LIN {X 0,Y 656.687,Z 491.433,A -85,B 0,C 180,E1 28585.458,E2 28585.458} C_VEL
LIN {X 0,Y 656.704,Z 491.397,A -85,B 0,C 180,E1 28582.346,E2 28582.346} C_VEL
LIN {X 0,Y 656.703,Z 491.421,A -85,B 0,C 180,E1 28580.485,E2 28580.485} C_VEL
LIN {X 0,Y 655.757,Z 491.547,A -85,B 0,C 180,E1 28579.813,E2 28579.813} C_VEL
LIN {X 0,Y 649.317,Z 492.327,A -85,B 0,C 180,E1 28577.929,E2 28577.929} C_VEL
LIN {X 0,Y 648.761,Z 492.387,A -85,B 0,C 180,E1 28577.439,E2 28577.439} C_VEL
LIN {X 0,Y 648.764,Z 492.41,A -85,B 0,C 180,E1 28574.279,E2 28574.279} C_VEL
LIN {X 0,Y 648.798,Z 492.658,A -85,B 0,C 180,E1 28571.504,E2 28571.504} C_VEL
LIN {X 0,Y 657.705,Z 514.386,A -85,B 0,C 180,E1 28569.164,E2 28569.164} C_VEL
LIN {X 0,Y 662.553,Z 527.138,A -85,B 0,C 180,E1 28567.894,E2 28567.894} C_VEL
LIN {X 0,Y 660.274,Z 574.159,A -85,B 0,C 180,E1 28564.707,E2 28564.707} C_VEL
LIN {X 0,Y 658.321,Z 619.289,A -85,B 0,C 180,E1 28561.727,E2 28561.727} C_VEL
LIN {X 0,Y 657.32,Z 647.28,A -85,B 0,C 180,E1 28559.941,E2 28559.941} C_VEL
LIN {X 0,Y 661.313,Z 670.225,A -85,B 0,C 180,E1 28559.432,E2 28559.432} C_VEL
LIN {X 0,Y 659.221,Z 900.56,A -85,B 0,C 180,E1 28556.758,E2 28556.758} C_VEL
LIN {X 0,Y 658.59,Z 956.878,A -85,B 0,C 180,E1 28556.077,E2 28556.077} C_VEL
LIN {X 0,Y 657.927,Z 978.152,A -85,B 0,C 180,E1 28555.662,E2 28555.662} C_VEL
LIN {X 0,Y 657.104,Z 999.966,A -85,B 0,C 180,E1 28555.073,E2 28555.073} C_VEL
LIN {X 0,Y 656.193,Z 1019.608,A -85,B 0,C 180,E1 28554.389,E2 28554.389} C_VEL
LIN {X 0,Y 655.097,Z 1039.619,A -85,B 0,C 180,E1 28553.523,E2 28553.523} C_VEL
LIN {X 0,Y 653.941,Z 1059.736,A -85,B 0,C 180,E1 28552.473,E2 28552.473} C_VEL
LIN {X 0,Y 652.846,Z 1078.181,A -85,B 0,C 180,E1 28551.33,E2 28551.33} C_VEL
LIN {X 0,Y 651.725,Z 1096.211,A -85,B 0,C 180,E1 28550.006,E2 28550.006} C_VEL
LIN {X 0,Y 650.802,Z 1113.681,A -85,B 0,C 180,E1 28548.543,E2 28548.543} C_VEL
LIN {X 0,Y 650.064,Z 1128.76,A -85,B 0,C 180,E1 28547.084,E2 28547.084} C_VEL
LIN {X 0,Y 649.402,Z 1143.252,A -85,B 0,C 180,E1 28545.448,E2 28545.448} C_VEL
LIN {X 0,Y 648.879,Z 1155.499,A -85,B 0,C 180,E1 28543.818,E2 28543.818} C_VEL
LIN {X 0,Y 648.48,Z 1167.039,A -85,B 0,C 180,E1 28542.014,E2 28542.014} C_VEL
LIN {X 0,Y 648.221,Z 1176.646,A -85,B 0,C 180,E1 28540.217,E2 28540.217} C_VEL
LIN {X 0,Y 648.06,Z 1184.7,A -85,B 0,C 180,E1 28538.339,E2 28538.339} C_VEL
LIN {X 0,Y 647.959,Z 1191.273,A -85,B 0,C 180,E1 28536.379,E2 28536.379} C_VEL
LIN {X 0,Y 647.926,Z 1195.934,A -85,B 0,C 180,E1 28534.495,E2 28534.495} C_VEL
LIN {X 0,Y 647.913,Z 1198.843,A -85,B 0,C 180,E1 28532.654,E2 28532.654} C_VEL
LIN {X 0,Y 647.907,Z 1200.334,A -85,B 0,C 180,E1 28530.619,E2 28530.619} C_VEL
LIN {X 0,Y 647.902,Z 1200.184,A -85,B 0,C 180,E1 28528.762,E2 28528.762} C_VEL
LIN {X 0,Y 647.911,Z 1198.323,A -85,B 0,C 180,E1 28526.851,E2 28526.851} C_VEL
LIN {X 0,Y 647.927,Z 1194.711,A -85,B 0,C 180,E1 28524.865,E2 28524.865} C_VEL
LIN {X 0,Y 647.972,Z 1189.734,A -85,B 0,C 180,E1 28522.998,E2 28522.998} C_VEL
LIN {X 0,Y 648.084,Z 1182.936,A -85,B 0,C 180,E1 28521.125,E2 28521.125} C_VEL
LIN {X 0,Y 648.283,Z 1174.365,A -85,B 0,C 180,E1 28519.244,E2 28519.244} C_VEL
LIN {X 0,Y 648.58,Z 1164.395,A -85,B 0,C 180,E1 28517.446,E2 28517.446} C_VEL
LIN {X 0,Y 648.996,Z 1152.865,A -85,B 0,C 180,E1 28515.717,E2 28515.717} C_VEL
LIN {X 0,Y 649.521,Z 1140.155,A -85,B 0,C 180,E1 28514.097,E2 28514.097} C_VEL
LIN {X 0,Y 650.186,Z 1126.103,A -85,B 0,C 180,E1 28512.55,E2 28512.55} C_VEL
LIN {X 0,Y 650.967,Z 1110.603,A -85,B 0,C 180,E1 28511.09,E2 28511.09} C_VEL
LIN {X 0,Y 652.128,Z 1089.891,A -85,B 0,C 180,E1 28509.414,E2 28509.414} C_VEL
LIN {X 0,Y 653.168,Z 1072.447,A -85,B 0,C 180,E1 28508.21,E2 28508.21} C_VEL
LIN {X 0,Y 654.338,Z 1053.073,A -85,B 0,C 180,E1 28507.067,E2 28507.067} C_VEL
LIN {X 0,Y 655.454,Z 1033.69,A -85,B 0,C 180,E1 28506.109,E2 28506.109} C_VEL
LIN {X 0,Y 656.48,Z 1013.299,A -85,B 0,C 180,E1 28505.287,E2 28505.287} C_VEL
LIN {X 0,Y 657.466,Z 991.151,A -85,B 0,C 180,E1 28504.578,E2 28504.578} C_VEL
LIN {X 0,Y 658.227,Z 970.127,A -85,B 0,C 180,E1 28504.069,E2 28504.069} C_VEL
LIN {X 0,Y 658.733,Z 948.225,A -85,B 0,C 180,E1 28503.712,E2 28503.712} C_VEL
LIN {X 0,Y 660.553,Z 758.083,A -85,B 0,C 180,E1 28501.489,E2 28501.489} C_VEL
LIN {X 0,Y 661.13,Z 667.999,A -85,B 0,C 180,E1 28500.44,E2 28500.44} C_VEL
LIN {X 0,Y 657.249,Z 646.305,A -85,B 0,C 180,E1 28499.93,E2 28499.93} C_VEL
LIN {X 0,Y 659.188,Z 599.058,A -85,B 0,C 180,E1 28496.857,E2 28496.857} C_VEL
LIN {X 0,Y 661.229,Z 553.533,A -85,B 0,C 180,E1 28493.814,E2 28493.814} C_VEL
LIN {X 0,Y 662.53,Z 526.699,A -85,B 0,C 180,E1 28491.981,E2 28491.981} C_VEL
LIN {X 0,Y 654.583,Z 506.578,A -85,B 0,C 180,E1 28489.933,E2 28489.933} C_VEL
LIN {X 0,Y 648.804,Z 492.683,A -85,B 0,C 180,E1 28488.4,E2 28488.4} C_VEL
LIN {X 0,Y 648.764,Z 492.389,A -85,B 0,C 180,E1 28486.417,E2 28486.417} C_VEL
LIN {X 0,Y 648.737,Z 492.391,A -85,B 0,C 180,E1 28483.305,E2 28483.305} C_VEL
LIN {X 0,Y 648.771,Z 492.42,A -85,B 0,C 180,E1 28480.282,E2 28480.282} C_VEL
LIN {X 0,Y 648.738,Z 492.392,A -85,B 0,C 180,E1 28477.17,E2 28477.17} C_VEL
LIN {X 0,Y 648.767,Z 492.414,A -85,B 0,C 180,E1 28474.125,E2 28474.125} C_VEL
LIN {X 0,Y 648.738,Z 492.415,A -85,B 0,C 180,E1 28470.984,E2 28470.984} C_VEL
LIN {X 0,Y 648.77,Z 492.416,A -85,B 0,C 180,E1 28467.939,E2 28467.939} C_VEL
LIN {X 0,Y 648.735,Z 492.417,A -85,B 0,C 180,E1 28464.786,E2 28464.786} C_VEL
LIN {X 0,Y 648.773,Z 492.416,A -85,B 0,C 180,E1 28461.709,E2 28461.709} C_VEL
LIN {X 0,Y 648.733,Z 492.407,A -85,B 0,C 180,E1 28458.583,E2 28458.583} C_VEL
LIN {X 0,Y 648.767,Z 492.41,A -85,B 0,C 180,E1 28455.556,E2 28455.556} C_VEL
LIN {X 0,Y 648.735,Z 492.416,A -85,B 0,C 180,E1 28452.461,E2 28452.461} C_VEL
LIN {X 0,Y 648.765,Z 492.411,A -85,B 0,C 180,E1 28449.403,E2 28449.403} C_VEL
LIN {X 0,Y 648.732,Z 492.408,A -85,B 0,C 180,E1 28446.283,E2 28446.283} C_VEL
LIN {X 0,Y 648.76,Z 492.423,A -85,B 0,C 180,E1 28443.269,E2 28443.269} C_VEL
LIN {X 0,Y 648.729,Z 492.412,A -85,B 0,C 180,E1 28440.088,E2 28440.088} C_VEL
LIN {X 0,Y 648.76,Z 492.41,A -85,B 0,C 180,E1 28437.085,E2 28437.085} C_VEL
LIN {X 0,Y 648.729,Z 492.416,A -85,B 0,C 180,E1 28433.895,E2 28433.895} C_VEL
LIN {X 0,Y 648.755,Z 492.41,A -85,B 0,C 180,E1 28430.955,E2 28430.955} C_VEL
LIN {X 0,Y 648.732,Z 492.407,A -85,B 0,C 180,E1 28427.81,E2 28427.81} C_VEL
LIN {X 0,Y 648.741,Z 492.422,A -85,B 0,C 180,E1 28424.902,E2 28424.902} C_VEL
LIN {X 0,Y 648.735,Z 492.415,A -85,B 0,C 180,E1 28421.674,E2 28421.674} C_VEL
LIN {X 0,Y 648.736,Z 492.411,A -85,B 0,C 180,E1 28418.764,E2 28418.764} C_VEL
LIN {X 0,Y 648.733,Z 492.407,A -85,B 0,C 180,E1 28415.505,E2 28415.505} C_VEL
LIN {X 0,Y 648.735,Z 492.423,A -85,B 0,C 180,E1 28412.592,E2 28412.592} C_VEL
LIN {X 0,Y 648.733,Z 492.416,A -85,B 0,C 180,E1 28409.318,E2 28409.318} C_VEL
LIN {X 0,Y 648.73,Z 492.385,A -85,B 0,C 180,E1 28406.404,E2 28406.404} C_VEL
LIN {X 0,Y 648.733,Z 492.417,A -85,B 0,C 180,E1 28403.161,E2 28403.161} C_VEL
LIN {X 0,Y 648.724,Z 492.39,A -85,B 0,C 180,E1 28400.272,E2 28400.272} C_VEL
LIN {X 0,Y 648.737,Z 492.398,A -85,B 0,C 180,E1 28397.058,E2 28397.058} C_VEL
LIN {X 0,Y 648.722,Z 492.426,A -85,B 0,C 180,E1 28394.159,E2 28394.159} C_VEL
LIN {X 0,Y 648.764,Z 492.635,A -85,B 0,C 180,E1 28391.933,E2 28391.933} C_VEL
LIN {X 0,Y 653.027,Z 502.897,A -85,B 0,C 180,E1 28390.827,E2 28390.827} C_VEL
LIN {X 0,Y 660.861,Z 521.597,A -85,B 0,C 180,E1 28388.95,E2 28388.95} C_VEL
LIN {X 0,Y 663.163,Z 527.795,A -85,B 0,C 180,E1 28388.368,E2 28388.368} C_VEL
LIN {X 0,Y 663.076,Z 532.792,A -85,B 0,C 180,E1 28388.071,E2 28388.071} C_VEL
LIN {X 0,Y 666.748,Z 551.518,A -85,B 0,C 180,E1 28387.604,E2 28387.604} C_VEL
LIN {X 0,Y 664.218,Z 791.043,A -85,B 0,C 180,E1 28384.694,E2 28384.694} C_VEL
LIN {X 0,Y 663.116,Z 920.342,A -85,B 0,C 180,E1 28383.165,E2 28383.165} C_VEL
LIN {X 0,Y 662.457,Z 946.043,A -85,B 0,C 180,E1 28382.706,E2 28382.706} C_VEL
LIN {X 0,Y 661.756,Z 967.211,A -85,B 0,C 180,E1 28382.199,E2 28382.199} C_VEL
LIN {X 0,Y 660.811,Z 989.286,A -85,B 0,C 180,E1 28381.518,E2 28381.518} C_VEL
LIN {X 0,Y 659.621,Z 1011.361,A -85,B 0,C 180,E1 28380.668,E2 28380.668} C_VEL
LIN {X 0,Y 658.378,Z 1033.294,A -85,B 0,C 180,E1 28379.675,E2 28379.675} C_VEL
LIN {X 0,Y 656.934,Z 1055.135,A -85,B 0,C 180,E1 28378.499,E2 28378.499} C_VEL
LIN {X 0,Y 655.615,Z 1075.664,A -85,B 0,C 180,E1 28377.227,E2 28377.227} C_VEL
LIN {X 0,Y 654.266,Z 1095.229,A -85,B 0,C 180,E1 28375.82,E2 28375.82} C_VEL
LIN {X 0,Y 653.063,Z 1113.21,A -85,B 0,C 180,E1 28374.357,E2 28374.357} C_VEL
LIN {X 0,Y 651.925,Z 1130.611,A -85,B 0,C 180,E1 28372.736,E2 28372.736} C_VEL
LIN {X 0,Y 650.985,Z 1145.636,A -85,B 0,C 180,E1 28371.158,E2 28371.158} C_VEL
LIN {X 0,Y 650.057,Z 1162.032,A -85,B 0,C 180,E1 28369.19,E2 28369.19} C_VEL
LIN {X 0,Y 649.427,Z 1174.524,A -85,B 0,C 180,E1 28367.471,E2 28367.471} C_VEL
LIN {X 0,Y 648.841,Z 1187.771,A -85,B 0,C 180,E1 28365.37,E2 28365.37} C_VEL
LIN {X 0,Y 648.474,Z 1197.565,A -85,B 0,C 180,E1 28363.554,E2 28363.554} C_VEL
LIN {X 0,Y 648.202,Z 1207.125,A -85,B 0,C 180,E1 28361.478,E2 28361.478} C_VEL
LIN {X 0,Y 648.054,Z 1214.515,A -85,B 0,C 180,E1 28359.502,E2 28359.502} C_VEL
LIN {X 0,Y 647.94,Z 1220.508,A -85,B 0,C 180,E1 28357.537,E2 28357.537} C_VEL
LIN {X 0,Y 647.901,Z 1225.336,A -85,B 0,C 180,E1 28355.402,E2 28355.402} C_VEL
LIN {X 0,Y 647.912,Z 1228.238,A -85,B 0,C 180,E1 28353.539,E2 28353.539} C_VEL
LIN {X 0,Y 647.904,Z 1230.169,A -85,B 0,C 180,E1 28351.326,E2 28351.326} C_VEL
LIN {X 0,Y 647.883,Z 1230.351,A -85,B 0,C 180,E1 28349.381,E2 28349.381} C_VEL
LIN {X 0,Y 647.899,Z 1229.361,A -85,B 0,C 180,E1 28347.523,E2 28347.523} C_VEL
LIN {X 0,Y 647.915,Z 1226.609,A -85,B 0,C 180,E1 28345.309,E2 28345.309} C_VEL
LIN {X 0,Y 647.941,Z 1222.896,A -85,B 0,C 180,E1 28343.443,E2 28343.443} C_VEL
LIN {X 0,Y 648.004,Z 1217.711,A -85,B 0,C 180,E1 28341.482,E2 28341.482} C_VEL
LIN {X 0,Y 648.138,Z 1210.307,A -85,B 0,C 180,E1 28339.331,E2 28339.331} C_VEL
LIN {X 0,Y 648.327,Z 1202.569,A -85,B 0,C 180,E1 28337.49,E2 28337.49} C_VEL
LIN {X 0,Y 648.682,Z 1191.897,A -85,B 0,C 180,E1 28335.358,E2 28335.358} C_VEL
LIN {X 0,Y 649.116,Z 1181.124,A -85,B 0,C 180,E1 28333.535,E2 28333.535} C_VEL
LIN {X 0,Y 649.762,Z 1168.129,A -85,B 0,C 180,E1 28331.612,E2 28331.612} C_VEL
LIN {X 0,Y 650.527,Z 1153.627,A -85,B 0,C 180,E1 28329.768,E2 28329.768} C_VEL
LIN {X 0,Y 651.499,Z 1137.653,A -85,B 0,C 180,E1 28327.971,E2 28327.971} C_VEL
LIN {X 0,Y 652.547,Z 1120.834,A -85,B 0,C 180,E1 28326.331,E2 28326.331} C_VEL
LIN {X 0,Y 653.8,Z 1102.507,A -85,B 0,C 180,E1 28324.743,E2 28324.743} C_VEL
LIN {X 0,Y 655.079,Z 1083.079,A -85,B 0,C 180,E1 28323.288,E2 28323.288} C_VEL
LIN {X 0,Y 656.509,Z 1062.412,A -85,B 0,C 180,E1 28321.927,E2 28321.927} C_VEL
LIN {X 0,Y 657.802,Z 1041.566,A -85,B 0,C 180,E1 28320.752,E2 28320.752} C_VEL
LIN {X 0,Y 659.216,Z 1019.235,A -85,B 0,C 180,E1 28319.664,E2 28319.664} C_VEL
LIN {X 0,Y 660.407,Z 996.993,A -85,B 0,C 180,E1 28318.765,E2 28318.765} C_VEL
LIN {X 0,Y 661.384,Z 976.854,A -85,B 0,C 180,E1 28318.08,E2 28318.08} C_VEL
LIN {X 0,Y 662.227,Z 952.701,A -85,B 0,C 180,E1 28317.437,E2 28317.437} C_VEL
LIN {X 0,Y 662.87,Z 930.275,A -85,B 0,C 180,E1 28316.993,E2 28316.993} C_VEL
LIN {X 0,Y 663.356,Z 902.806,A -85,B 0,C 180,E1 28316.61,E2 28316.61} C_VEL
LIN {X 0,Y 665.273,Z 677.94,A -85,B 0,C 180,E1 28313.952,E2 28313.952} C_VEL
LIN {X 0,Y 666.596,Z 549.747,A -85,B 0,C 180,E1 28312.364,E2 28312.364} C_VEL
LIN {X 0,Y 662.988,Z 531.826,A -85,B 0,C 180,E1 28311.889,E2 28311.889} C_VEL
LIN {X 0,Y 663.187,Z 527.295,A -85,B 0,C 180,E1 28311.6,E2 28311.6} C_VEL
LIN {X 0,Y 654.413,Z 506.148,A -85,B 0,C 180,E1 28309.508,E2 28309.508} C_VEL
LIN {X 0,Y 648.773,Z 492.677,A -85,B 0,C 180,E1 28308.078,E2 28308.078} C_VEL
LIN {X 0,Y 648.772,Z 492.403,A -85,B 0,C 180,E1 28306.579,E2 28306.579} C_VEL
LIN {X 0,Y 648.71,Z 492.393,A -85,B 0,C 180,E1 28303.55,E2 28303.55} C_VEL
LIN {X 0,Y 648.77,Z 492.407,A -85,B 0,C 180,E1 28300.571,E2 28300.571} C_VEL
LIN {X 0,Y 648.718,Z 492.415,A -85,B 0,C 180,E1 28297.462,E2 28297.462} C_VEL
LIN {X 0,Y 648.755,Z 492.399,A -85,B 0,C 180,E1 28294.554,E2 28294.554} C_VEL
LIN {X 0,Y 648.724,Z 492.417,A -85,B 0,C 180,E1 28291.366,E2 28291.366} C_VEL
LIN {X 0,Y 648.751,Z 492.409,A -85,B 0,C 180,E1 28288.441,E2 28288.441} C_VEL
LIN {X 0,Y 648.732,Z 492.411,A -85,B 0,C 180,E1 28285.274,E2 28285.274} C_VEL
LIN {X 0,Y 648.741,Z 492.415,A -85,B 0,C 180,E1 28282.372,E2 28282.372} C_VEL
LIN {X 0,Y 648.738,Z 492.421,A -85,B 0,C 180,E1 28279.131,E2 28279.131} C_VEL
LIN {X 0,Y 648.742,Z 492.408,A -85,B 0,C 180,E1 28276.199,E2 28276.199} C_VEL
LIN {X 0,Y 648.742,Z 492.41,A -85,B 0,C 180,E1 28273.004,E2 28273.004} C_VEL
LIN {X 0,Y 648.747,Z 492.414,A -85,B 0,C 180,E1 28269.992,E2 28269.992} C_VEL
LIN {X 0,Y 648.746,Z 492.42,A -85,B 0,C 180,E1 28266.816,E2 28266.816} C_VEL
LIN {X 0,Y 648.747,Z 492.405,A -85,B 0,C 180,E1 28263.8,E2 28263.8} C_VEL
LIN {X 0,Y 648.747,Z 492.417,A -85,B 0,C 180,E1 28260.618,E2 28260.618} C_VEL
LIN {X 0,Y 648.75,Z 492.41,A -85,B 0,C 180,E1 28257.615,E2 28257.615} C_VEL
LIN {X 0,Y 648.745,Z 492.409,A -85,B 0,C 180,E1 28254.428,E2 28254.428} C_VEL
LIN {X 0,Y 648.756,Z 492.413,A -85,B 0,C 180,E1 28251.402,E2 28251.402} C_VEL
LIN {X 0,Y 648.743,Z 492.422,A -85,B 0,C 180,E1 28248.171,E2 28248.171} C_VEL
LIN {X 0,Y 648.77,Z 492.401,A -85,B 0,C 180,E1 28245.084,E2 28245.084} C_VEL
LIN {X 0,Y 648.743,Z 492.412,A -85,B 0,C 180,E1 28241.953,E2 28241.953} C_VEL
LIN {X 0,Y 648.77,Z 492.413,A -85,B 0,C 180,E1 28238.86,E2 28238.86} C_VEL
LIN {X 0,Y 648.741,Z 492.421,A -85,B 0,C 180,E1 28235.699,E2 28235.699} C_VEL
LIN {X 0,Y 648.766,Z 492.406,A -85,B 0,C 180,E1 28232.659,E2 28232.659} C_VEL
LIN {X 0,Y 648.743,Z 492.415,A -85,B 0,C 180,E1 28229.53,E2 28229.53} C_VEL
LIN {X 0,Y 648.766,Z 492.408,A -85,B 0,C 180,E1 28226.488,E2 28226.488} C_VEL
LIN {X 0,Y 648.744,Z 492.399,A -85,B 0,C 180,E1 28223.382,E2 28223.382} C_VEL
LIN {X 0,Y 648.768,Z 492.41,A -85,B 0,C 180,E1 28220.268,E2 28220.268} C_VEL
LIN {X 0,Y 648.761,Z 492.387,A -85,B 0,C 180,E1 28217.439,E2 28217.439} C_VEL
LIN {X 0,Y 647.741,Z 492.518,A -85,B 0,C 180,E1 28216.759,E2 28216.759} C_VEL
LIN {X 0,Y 641.323,Z 493.349,A -85,B 0,C 180,E1 28214.852,E2 28214.852} C_VEL
LIN {X 0,Y 640.821,Z 493.4,A -85,B 0,C 180,E1 28214.356,E2 28214.356} C_VEL
LIN {X 0,Y 640.86,Z 493.629,A -85,B 0,C 180,E1 28212.067,E2 28212.067} C_VEL
LIN {X 0,Y 645.223,Z 504.16,A -85,B 0,C 180,E1 28210.865,E2 28210.865} C_VEL
LIN {X 0,Y 653.936,Z 525.683,A -85,B 0,C 180,E1 28208.596,E2 28208.596} C_VEL
LIN {X 0,Y 655.646,Z 530.796,A -85,B 0,C 180,E1 28208.101,E2 28208.101} C_VEL
LIN {X 0,Y 653.146,Z 578.763,A -85,B 0,C 180,E1 28204.82,E2 28204.82} C_VEL
LIN {X 0,Y 651.038,Z 624.276,A -85,B 0,C 180,E1 28201.788,E2 28201.788} C_VEL
LIN {X 0,Y 650.196,Z 646.313,A -85,B 0,C 180,E1 28200.37,E2 28200.37} C_VEL
LIN {X 0,Y 654.607,Z 671.415,A -85,B 0,C 180,E1 28199.802,E2 28199.802} C_VEL
LIN {X 0,Y 652.343,Z 919.767,A -85,B 0,C 180,E1 28196.919,E2 28196.919} C_VEL
LIN {X 0,Y 651.813,Z 958.309,A -85,B 0,C 180,E1 28196.435,E2 28196.435} C_VEL
LIN {X 0,Y 651.111,Z 979.366,A -85,B 0,C 180,E1 28196.015,E2 28196.015} C_VEL
LIN {X 0,Y 650.23,Z 1000.616,A -85,B 0,C 180,E1 28195.43,E2 28195.43} C_VEL
LIN {X 0,Y 649.223,Z 1020.828,A -85,B 0,C 180,E1 28194.717,E2 28194.717} C_VEL
LIN {X 0,Y 648.016,Z 1040.55,A -85,B 0,C 180,E1 28193.844,E2 28193.844} C_VEL
LIN {X 0,Y 646.736,Z 1060.42,A -85,B 0,C 180,E1 28192.785,E2 28192.785} C_VEL
LIN {X 0,Y 645.476,Z 1079.395,A -85,B 0,C 180,E1 28191.586,E2 28191.586} C_VEL
LIN {X 0,Y 644.291,Z 1096.703,A -85,B 0,C 180,E1 28190.294,E2 28190.294} C_VEL
LIN {X 0,Y 643.211,Z 1113.172,A -85,B 0,C 180,E1 28188.864,E2 28188.864} C_VEL
LIN {X 0,Y 642.272,Z 1128.765,A -85,B 0,C 180,E1 28187.298,E2 28187.298} C_VEL
LIN {X 0,Y 641.549,Z 1143.255,A -85,B 0,C 180,E1 28185.642,E2 28185.642} C_VEL
LIN {X 0,Y 640.981,Z 1155.501,A -85,B 0,C 180,E1 28183.992,E2 28183.992} C_VEL
LIN {X 0,Y 640.54,Z 1167.041,A -85,B 0,C 180,E1 28182.165,E2 28182.165} C_VEL
LIN {X 0,Y 640.254,Z 1176.649,A -85,B 0,C 180,E1 28180.346,E2 28180.346} C_VEL
LIN {X 0,Y 640.078,Z 1184.703,A -85,B 0,C 180,E1 28178.444,E2 28178.444} C_VEL
LIN {X 0,Y 639.962,Z 1191.274,A -85,B 0,C 180,E1 28176.459,E2 28176.459} C_VEL
LIN {X 0,Y 639.925,Z 1195.988,A -85,B 0,C 180,E1 28174.521,E2 28174.521} C_VEL
LIN {X 0,Y 639.912,Z 1198.843,A -85,B 0,C 180,E1 28172.687,E2 28172.687} C_VEL
LIN {X 0,Y 639.907,Z 1200.334,A -85,B 0,C 180,E1 28170.627,E2 28170.627} C_VEL
LIN {X 0,Y 639.902,Z 1200.184,A -85,B 0,C 180,E1 28168.747,E2 28168.747} C_VEL
LIN {X 0,Y 639.911,Z 1198.349,A -85,B 0,C 180,E1 28166.833,E2 28166.833} C_VEL
LIN {X 0,Y 639.931,Z 1194.71,A -85,B 0,C 180,E1 28164.801,E2 28164.801} C_VEL
LIN {X 0,Y 639.982,Z 1189.732,A -85,B 0,C 180,E1 28162.91,E2 28162.91} C_VEL
LIN {X 0,Y 640.103,Z 1182.934,A -85,B 0,C 180,E1 28161.013,E2 28161.013} C_VEL
LIN {X 0,Y 640.319,Z 1174.362,A -85,B 0,C 180,E1 28159.109,E2 28159.109} C_VEL
LIN {X 0,Y 640.651,Z 1164.361,A -85,B 0,C 180,E1 28157.283,E2 28157.283} C_VEL
LIN {X 0,Y 641.1,Z 1152.947,A -85,B 0,C 180,E1 28155.55,E2 28155.55} C_VEL
LIN {X 0,Y 641.681,Z 1140.149,A -85,B 0,C 180,E1 28153.898,E2 28153.898} C_VEL
LIN {X 0,Y 642.459,Z 1125.255,A -85,B 0,C 180,E1 28152.24,E2 28152.24} C_VEL
LIN {X 0,Y 643.442,Z 1109.685,A -85,B 0,C 180,E1 28150.719,E2 28150.719} C_VEL
LIN {X 0,Y 644.535,Z 1093.11,A -85,B 0,C 180,E1 28149.334,E2 28149.334} C_VEL
LIN {X 0,Y 645.789,Z 1074.445,A -85,B 0,C 180,E1 28147.995,E2 28147.995} C_VEL
LIN {X 0,Y 647.09,Z 1055.489,A -85,B 0,C 180,E1 28146.839,E2 28146.839} C_VEL
LIN {X 0,Y 648.263,Z 1036.558,A -85,B 0,C 180,E1 28145.875,E2 28145.875} C_VEL
LIN {X 0,Y 649.469,Z 1015.731,A -85,B 0,C 180,E1 28145.002,E2 28145.002} C_VEL
LIN {X 0,Y 650.499,Z 995.068,A -85,B 0,C 180,E1 28144.307,E2 28144.307} C_VEL
LIN {X 0,Y 651.297,Z 974.495,A -85,B 0,C 180,E1 28143.785,E2 28143.785} C_VEL
LIN {X 0,Y 651.929,Z 951.776,A -85,B 0,C 180,E1 28143.38,E2 28143.38} C_VEL
LIN {X 0,Y 653.583,Z 787.252,A -85,B 0,C 180,E1 28141.444,E2 28141.444} C_VEL
LIN {X 0,Y 654.426,Z 669.373,A -85,B 0,C 180,E1 28140.073,E2 28140.073} C_VEL
LIN {X 0,Y 650.137,Z 645.401,A -85,B 0,C 180,E1 28139.502,E2 28139.502} C_VEL
LIN {X 0,Y 652.213,Z 598.269,A -85,B 0,C 180,E1 28136.398,E2 28136.398} C_VEL
LIN {X 0,Y 654.413,Z 553.495,A -85,B 0,C 180,E1 28133.371,E2 28133.371} C_VEL
LIN {X 0,Y 655.594,Z 529.964,A -85,B 0,C 180,E1 28131.743,E2 28131.743} C_VEL
LIN {X 0,Y 646.809,Z 507.86,A -85,B 0,C 180,E1 28129.447,E2 28129.447} C_VEL
LIN {X 0,Y 640.888,Z 493.793,A -85,B 0,C 180,E1 28127.868,E2 28127.868} C_VEL
LIN {X 0,Y 640.794,Z 493.374,A -85,B 0,C 180,E1 28127.303,E2 28127.303} C_VEL
LIN {X 0,Y 640.826,Z 493.394,A -85,B 0,C 180,E1 28124.224,E2 28124.224} C_VEL
LIN {X 0,Y 640.795,Z 493.403,A -85,B 0,C 180,E1 28121.093,E2 28121.093} C_VEL
LIN {X 0,Y 640.824,Z 493.37,A -85,B 0,C 180,E1 28118.049,E2 28118.049} C_VEL
LIN {X 0,Y 640.794,Z 493.408,A -85,B 0,C 180,E1 28114.936,E2 28114.936} C_VEL
LIN {X 0,Y 640.828,Z 493.409,A -85,B 0,C 180,E1 28111.921,E2 28111.921} C_VEL
LIN {X 0,Y 640.795,Z 493.406,A -85,B 0,C 180,E1 28108.827,E2 28108.827} C_VEL
LIN {X 0,Y 640.83,Z 493.403,A -85,B 0,C 180,E1 28105.806,E2 28105.806} C_VEL
LIN {X 0,Y 640.793,Z 493.395,A -85,B 0,C 180,E1 28102.67,E2 28102.67} C_VEL
LIN {X 0,Y 640.829,Z 493.398,A -85,B 0,C 180,E1 28099.696,E2 28099.696} C_VEL
LIN {X 0,Y 640.798,Z 493.405,A -85,B 0,C 180,E1 28096.592,E2 28096.592} C_VEL
LIN {X 0,Y 640.828,Z 493.402,A -85,B 0,C 180,E1 28093.536,E2 28093.536} C_VEL
LIN {X 0,Y 640.796,Z 493.392,A -85,B 0,C 180,E1 28090.428,E2 28090.428} C_VEL
LIN {X 0,Y 640.822,Z 493.408,A -85,B 0,C 180,E1 28087.441,E2 28087.441} C_VEL
LIN {X 0,Y 640.799,Z 493.403,A -85,B 0,C 180,E1 28084.295,E2 28084.295} C_VEL
LIN {X 0,Y 640.818,Z 493.397,A -85,B 0,C 180,E1 28081.252,E2 28081.252} C_VEL
LIN {X 0,Y 640.797,Z 493.403,A -85,B 0,C 180,E1 28078.122,E2 28078.122} C_VEL
LIN {X 0,Y 640.816,Z 493.403,A -85,B 0,C 180,E1 28075.077,E2 28075.077} C_VEL
LIN {X 0,Y 640.794,Z 493.391,A -85,B 0,C 180,E1 28071.927,E2 28071.927} C_VEL
LIN {X 0,Y 640.813,Z 493.41,A -85,B 0,C 180,E1 28068.935,E2 28068.935} C_VEL
LIN {X 0,Y 640.79,Z 493.405,A -85,B 0,C 180,E1 28065.727,E2 28065.727} C_VEL
LIN {X 0,Y 640.809,Z 493.398,A -85,B 0,C 180,E1 28062.754,E2 28062.754} C_VEL
LIN {X 0,Y 640.79,Z 493.398,A -85,B 0,C 180,E1 28059.541,E2 28059.541} C_VEL
LIN {X 0,Y 640.803,Z 493.411,A -85,B 0,C 180,E1 28056.651,E2 28056.651} C_VEL
LIN {X 0,Y 640.793,Z 493.406,A -85,B 0,C 180,E1 28053.39,E2 28053.39} C_VEL
LIN {X 0,Y 640.801,Z 493.406,A -85,B 0,C 180,E1 28050.457,E2 28050.457} C_VEL
LIN {X 0,Y 640.787,Z 493.375,A -85,B 0,C 180,E1 28047.217,E2 28047.217} C_VEL
LIN {X 0,Y 640.799,Z 493.406,A -85,B 0,C 180,E1 28044.297,E2 28044.297} C_VEL
LIN {X 0,Y 640.783,Z 493.371,A -85,B 0,C 180,E1 28041.035,E2 28041.035} C_VEL
LIN {X 0,Y 640.789,Z 493.414,A -85,B 0,C 180,E1 28038.218,E2 28038.218} C_VEL
LIN {X 0,Y 640.795,Z 493.392,A -85,B 0,C 180,E1 28034.978,E2 28034.978} C_VEL
LIN {X 0,Y 640.799,Z 493.589,A -85,B 0,C 180,E1 28032.502,E2 28032.502} C_VEL
LIN {X 0,Y 641.926,Z 496.622,A -85,B 0,C 180,E1 28032.146,E2 28032.146} C_VEL
LIN {X 0,Y 650.144,Z 515.394,A -85,B 0,C 180,E1 28030.149,E2 28030.149} C_VEL
LIN {X 0,Y 656.315,Z 530.866,A -85,B 0,C 180,E1 28028.623,E2 28028.623} C_VEL
LIN {X 0,Y 656.391,Z 534.026,A -85,B 0,C 180,E1 28028.455,E2 28028.455} C_VEL
LIN {X 0,Y 660.104,Z 553.023,A -85,B 0,C 180,E1 28027.975,E2 28027.975} C_VEL
LIN {X 0,Y 657.263,Z 788.968,A -85,B 0,C 180,E1 28025.06,E2 28025.06} C_VEL
LIN {X 0,Y 655.972,Z 920.648,A -85,B 0,C 180,E1 28023.477,E2 28023.477} C_VEL
LIN {X 0,Y 655.269,Z 946.268,A -85,B 0,C 180,E1 28023.013,E2 28023.013} C_VEL
LIN {X 0,Y 654.509,Z 967.887,A -85,B 0,C 180,E1 28022.488,E2 28022.488} C_VEL
LIN {X 0,Y 653.447,Z 993.177,A -85,B 0,C 180,E1 28021.703,E2 28021.703} C_VEL
LIN {X 0,Y 652.476,Z 1013.342,A -85,B 0,C 180,E1 28020.939,E2 28020.939} C_VEL
LIN {X 0,Y 651.301,Z 1033.298,A -85,B 0,C 180,E1 28020.031,E2 28020.031} C_VEL
LIN {X 0,Y 649.752,Z 1055.13,A -85,B 0,C 180,E1 28018.844,E2 28018.844} C_VEL
LIN {X 0,Y 648.312,Z 1075.667,A -85,B 0,C 180,E1 28017.56,E2 28017.56} C_VEL
LIN {X 0,Y 646.863,Z 1095.227,A -85,B 0,C 180,E1 28016.137,E2 28016.137} C_VEL
LIN {X 0,Y 645.554,Z 1113.071,A -85,B 0,C 180,E1 28014.671,E2 28014.671} C_VEL
LIN {X 0,Y 644.312,Z 1130.61,A -85,B 0,C 180,E1 28013.02,E2 28013.02} C_VEL
LIN {X 0,Y 643.278,Z 1145.866,A -85,B 0,C 180,E1 28011.398,E2 28011.398} C_VEL
LIN {X 0,Y 642.296,Z 1161.824,A -85,B 0,C 180,E1 28009.459,E2 28009.459} C_VEL
LIN {X 0,Y 641.577,Z 1174.522,A -85,B 0,C 180,E1 28007.692,E2 28007.692} C_VEL
LIN {X 0,Y 640.935,Z 1187.772,A -85,B 0,C 180,E1 28005.564,E2 28005.564} C_VEL
LIN {X 0,Y 640.537,Z 1197.564,A -85,B 0,C 180,E1 28003.725,E2 28003.725} C_VEL
LIN {X 0,Y 640.242,Z 1207.126,A -85,B 0,C 180,E1 28001.622,E2 28001.622} C_VEL
LIN {X 0,Y 640.062,Z 1214.515,A -85,B 0,C 180,E1 27999.622,E2 27999.622} C_VEL
LIN {X 0,Y 639.95,Z 1220.508,A -85,B 0,C 180,E1 27997.632,E2 27997.632} C_VEL
LIN {X 0,Y 639.905,Z 1225.336,A -85,B 0,C 180,E1 27995.469,E2 27995.469} C_VEL
LIN {X 0,Y 639.912,Z 1228.238,A -85,B 0,C 180,E1 27993.583,E2 27993.583} C_VEL
LIN {X 0,Y 639.903,Z 1230.169,A -85,B 0,C 180,E1 27991.343,E2 27991.343} C_VEL
LIN {X 0,Y 639.883,Z 1230.35,A -85,B 0,C 180,E1 27989.373,E2 27989.373} C_VEL
LIN {X 0,Y 639.897,Z 1229.361,A -85,B 0,C 180,E1 27987.492,E2 27987.492} C_VEL
LIN {X 0,Y 639.912,Z 1226.61,A -85,B 0,C 180,E1 27985.25,E2 27985.25} C_VEL
LIN {X 0,Y 639.945,Z 1222.896,A -85,B 0,C 180,E1 27983.361,E2 27983.361} C_VEL
LIN {X 0,Y 640.009,Z 1217.711,A -85,B 0,C 180,E1 27981.374,E2 27981.374} C_VEL
LIN {X 0,Y 640.157,Z 1210.31,A -85,B 0,C 180,E1 27979.197,E2 27979.197} C_VEL
LIN {X 0,Y 640.369,Z 1202.753,A -85,B 0,C 180,E1 27977.374,E2 27977.374} C_VEL
LIN {X 0,Y 640.747,Z 1192.41,A -85,B 0,C 180,E1 27975.265,E2 27975.265} C_VEL
LIN {X 0,Y 641.239,Z 1181.123,A -85,B 0,C 180,E1 27973.327,E2 27973.327} C_VEL
LIN {X 0,Y 641.945,Z 1168.128,A -85,B 0,C 180,E1 27971.38,E2 27971.38} C_VEL
LIN {X 0,Y 642.79,Z 1153.625,A -85,B 0,C 180,E1 27969.514,E2 27969.514} C_VEL
LIN {X 0,Y 643.823,Z 1138.007,A -85,B 0,C 180,E1 27967.733,E2 27967.733} C_VEL
LIN {X 0,Y 644.994,Z 1120.834,A -85,B 0,C 180,E1 27966.037,E2 27966.037} C_VEL
LIN {X 0,Y 646.34,Z 1102.508,A -85,B 0,C 180,E1 27964.431,E2 27964.431} C_VEL
LIN {X 0,Y 647.747,Z 1083.049,A -85,B 0,C 180,E1 27962.96,E2 27962.96} C_VEL
LIN {X 0,Y 649.224,Z 1063.177,A -85,B 0,C 180,E1 27961.633,E2 27961.633} C_VEL
LIN {X 0,Y 650.635,Z 1042.29,A -85,B 0,C 180,E1 27960.439,E2 27960.439} C_VEL
LIN {X 0,Y 651.976,Z 1022.236,A -85,B 0,C 180,E1 27959.444,E2 27959.444} C_VEL
LIN {X 0,Y 653.157,Z 999.802,A -85,B 0,C 180,E1 27958.533,E2 27958.533} C_VEL
LIN {X 0,Y 654.077,Z 978.978,A -85,B 0,C 180,E1 27957.835,E2 27957.835} C_VEL
LIN {X 0,Y 654.974,Z 955.303,A -85,B 0,C 180,E1 27957.185,E2 27957.185} C_VEL
LIN {X 0,Y 655.672,Z 931.683,A -85,B 0,C 180,E1 27956.703,E2 27956.703} C_VEL
LIN {X 0,Y 656.203,Z 906.757,A -85,B 0,C 180,E1 27956.336,E2 27956.336} C_VEL
LIN {X 0,Y 658.409,Z 681.268,A -85,B 0,C 180,E1 27953.629,E2 27953.629} C_VEL
LIN {X 0,Y 659.962,Z 551.351,A -85,B 0,C 180,E1 27951.994,E2 27951.994} C_VEL
LIN {X 0,Y 656.245,Z 532.953,A -85,B 0,C 180,E1 27951.506,E2 27951.506} C_VEL
LIN {X 0,Y 656.21,Z 530.422,A -85,B 0,C 180,E1 27951.339,E2 27951.339} C_VEL
LIN {X 0,Y 646.982,Z 508.07,A -85,B 0,C 180,E1 27949.09,E2 27949.09} C_VEL
LIN {X 0,Y 640.811,Z 493.667,A -85,B 0,C 180,E1 27947.517,E2 27947.517} C_VEL
LIN {X 0,Y 640.809,Z 493.407,A -85,B 0,C 180,E1 27946.128,E2 27946.128} C_VEL
LIN {X 0,Y 640.777,Z 493.382,A -85,B 0,C 180,E1 27943.223,E2 27943.223} C_VEL
LIN {X 0,Y 640.829,Z 493.38,A -85,B 0,C 180,E1 27940.122,E2 27940.122} C_VEL
LIN {X 0,Y 640.779,Z 493.408,A -85,B 0,C 180,E1 27937.122,E2 27937.122} C_VEL
LIN {X 0,Y 640.827,Z 493.372,A -85,B 0,C 180,E1 27934.055,E2 27934.055} C_VEL
LIN {X 0,Y 640.778,Z 493.407,A -85,B 0,C 180,E1 27931.058,E2 27931.058} C_VEL
LIN {X 0,Y 640.834,Z 493.396,A -85,B 0,C 180,E1 27928.113,E2 27928.113} C_VEL
LIN {X 0,Y 640.781,Z 493.399,A -85,B 0,C 180,E1 27925.016,E2 27925.016} C_VEL
LIN {X 0,Y 640.836,Z 493.404,A -85,B 0,C 180,E1 27921.992,E2 27921.992} C_VEL
LIN {X 0,Y 640.787,Z 493.409,A -85,B 0,C 180,E1 27918.939,E2 27918.939} C_VEL
LIN {X 0,Y 640.826,Z 493.396,A -85,B 0,C 180,E1 27915.939,E2 27915.939} C_VEL
LIN {X 0,Y 640.789,Z 493.397,A -85,B 0,C 180,E1 27912.782,E2 27912.782} C_VEL
LIN {X 0,Y 640.825,Z 493.402,A -85,B 0,C 180,E1 27909.792,E2 27909.792} C_VEL
LIN {X 0,Y 640.793,Z 493.409,A -85,B 0,C 180,E1 27906.631,E2 27906.631} C_VEL
LIN {X 0,Y 640.825,Z 493.392,A -85,B 0,C 180,E1 27903.578,E2 27903.578} C_VEL
LIN {X 0,Y 640.795,Z 493.404,A -85,B 0,C 180,E1 27900.447,E2 27900.447} C_VEL
LIN {X 0,Y 640.826,Z 493.398,A -85,B 0,C 180,E1 27897.407,E2 27897.407} C_VEL
LIN {X 0,Y 640.797,Z 493.398,A -85,B 0,C 180,E1 27894.269,E2 27894.269} C_VEL
LIN {X 0,Y 640.83,Z 493.402,A -85,B 0,C 180,E1 27891.204,E2 27891.204} C_VEL
LIN {X 0,Y 640.797,Z 493.409,A -85,B 0,C 180,E1 27888.022,E2 27888.022} C_VEL
LIN {X 0,Y 640.832,Z 493.39,A -85,B 0,C 180,E1 27884.97,E2 27884.97} C_VEL
LIN {X 0,Y 640.797,Z 493.399,A -85,B 0,C 180,E1 27881.815,E2 27881.815} C_VEL
LIN {X 0,Y 640.831,Z 493.403,A -85,B 0,C 180,E1 27878.777,E2 27878.777} C_VEL
LIN {X 0,Y 640.801,Z 493.41,A -85,B 0,C 180,E1 27875.673,E2 27875.673} C_VEL
LIN {X 0,Y 640.829,Z 493.395,A -85,B 0,C 180,E1 27872.594,E2 27872.594} C_VEL
LIN {X 0,Y 640.802,Z 493.404,A -85,B 0,C 180,E1 27869.462,E2 27869.462} C_VEL
LIN {X 0,Y 640.826,Z 493.397,A -85,B 0,C 180,E1 27866.364,E2 27866.364} C_VEL
LIN {X 0,Y 640.801,Z 493.385,A -85,B 0,C 180,E1 27863.3,E2 27863.3} C_VEL
LIN {X 0,Y 640.828,Z 493.4,A -85,B 0,C 180,E1 27860.228,E2 27860.228} C_VEL
LIN {X 0,Y 640.803,Z 493.374,A -85,B 0,C 180,E1 27857.131,E2 27857.131} C_VEL
LIN {X 0,Y 640.821,Z 493.4,A -85,B 0,C 180,E1 27854.356,E2 27854.356} C_VEL
LIN {X 0,Y 639.957,Z 493.502,A -85,B 0,C 180,E1 27853.937,E2 27853.937} C_VEL
LIN {X 0,Y 634.781,Z 494.431,A -85,B 0,C 180,E1 27852.978,E2 27852.978} C_VEL
LIN {X 0,Y 633.571,Z 495.611,A -85,B 0,C 180,E1 27852.606,E2 27852.606} C_VEL
LIN {X 0,Y 633.832,Z 497.267,A -85,B 0,C 180,E1 27852.321,E2 27852.321} C_VEL
LIN {X 0,Y 641.987,Z 516.276,A -85,B 0,C 180,E1 27850.179,E2 27850.179} C_VEL
LIN {X 0,Y 648.784,Z 533.779,A -85,B 0,C 180,E1 27848.359,E2 27848.359} C_VEL
LIN {X 0,Y 646.133,Z 581.095,A -85,B 0,C 180,E1 27845.091,E2 27845.091} C_VEL
LIN {X 0,Y 643.852,Z 626.83,A -85,B 0,C 180,E1 27842.013,E2 27842.013} C_VEL
LIN {X 0,Y 643.115,Z 645.489,A -85,B 0,C 180,E1 27840.805,E2 27840.805} C_VEL
LIN {X 0,Y 647.93,Z 672.788,A -85,B 0,C 180,E1 27840.178,E2 27840.178} C_VEL
LIN {X 0,Y 645.63,Z 920.642,A -85,B 0,C 180,E1 27837.296,E2 27837.296} C_VEL
LIN {X 0,Y 645.14,Z 957.989,A -85,B 0,C 180,E1 27836.833,E2 27836.833} C_VEL
LIN {X 0,Y 644.406,Z 978.805,A -85,B 0,C 180,E1 27836.418,E2 27836.418} C_VEL
LIN {X 0,Y 643.427,Z 1000.643,A -85,B 0,C 180,E1 27835.817,E2 27835.817} C_VEL
LIN {X 0,Y 642.339,Z 1020.833,A -85,B 0,C 180,E1 27835.098,E2 27835.098} C_VEL
LIN {X 0,Y 641.027,Z 1040.589,A -85,B 0,C 180,E1 27834.219,E2 27834.219} C_VEL
LIN {X 0,Y 639.64,Z 1060.48,A -85,B 0,C 180,E1 27833.15,E2 27833.15} C_VEL
LIN {X 0,Y 638.272,Z 1079.052,A -85,B 0,C 180,E1 27831.966,E2 27831.966} C_VEL
LIN {X 0,Y 636.925,Z 1096.635,A -85,B 0,C 180,E1 27830.636,E2 27830.636} C_VEL
LIN {X 0,Y 635.684,Z 1113.479,A -85,B 0,C 180,E1 27829.154,E2 27829.154} C_VEL
LIN {X 0,Y 634.647,Z 1128.737,A -85,B 0,C 180,E1 27827.601,E2 27827.601} C_VEL
LIN {X 0,Y 633.771,Z 1142.783,A -85,B 0,C 180,E1 27825.933,E2 27825.933} C_VEL
LIN {X 0,Y 633.029,Z 1156.775,A -85,B 0,C 180,E1 27823.985,E2 27823.985} C_VEL
LIN {X 0,Y 632.585,Z 1167.558,A -85,B 0,C 180,E1 27822.228,E2 27822.228} C_VEL
LIN {X 0,Y 632.275,Z 1177.106,A -85,B 0,C 180,E1 27820.376,E2 27820.376} C_VEL
LIN {X 0,Y 632.094,Z 1184.705,A -85,B 0,C 180,E1 27818.551,E2 27818.551} C_VEL
LIN {X 0,Y 631.965,Z 1191.276,A -85,B 0,C 180,E1 27816.541,E2 27816.541} C_VEL
LIN {X 0,Y 631.922,Z 1195.9,A -85,B 0,C 180,E1 27814.628,E2 27814.628} C_VEL
LIN {X 0,Y 631.912,Z 1198.843,A -85,B 0,C 180,E1 27812.721,E2 27812.721} C_VEL
LIN {X 0,Y 631.907,Z 1200.333,A -85,B 0,C 180,E1 27810.635,E2 27810.635} C_VEL
LIN {X 0,Y 631.901,Z 1200.184,A -85,B 0,C 180,E1 27808.731,E2 27808.731} C_VEL
LIN {X 0,Y 631.91,Z 1198.376,A -85,B 0,C 180,E1 27806.815,E2 27806.815} C_VEL
LIN {X 0,Y 631.934,Z 1194.708,A -85,B 0,C 180,E1 27804.735,E2 27804.735} C_VEL
LIN {X 0,Y 631.994,Z 1189.73,A -85,B 0,C 180,E1 27802.82,E2 27802.82} C_VEL
LIN {X 0,Y 632.125,Z 1182.932,A -85,B 0,C 180,E1 27800.899,E2 27800.899} C_VEL
LIN {X 0,Y 632.355,Z 1174.359,A -85,B 0,C 180,E1 27798.97,E2 27798.97} C_VEL
LIN {X 0,Y 632.722,Z 1164.386,A -85,B 0,C 180,E1 27797.126,E2 27797.126} C_VEL
LIN {X 0,Y 633.214,Z 1152.943,A -85,B 0,C 180,E1 27795.366,E2 27795.366} C_VEL
LIN {X 0,Y 633.94,Z 1139.747,A -85,B 0,C 180,E1 27793.601,E2 27793.601} C_VEL
LIN {X 0,Y 634.878,Z 1125.159,A -85,B 0,C 180,E1 27791.926,E2 27791.926} C_VEL
LIN {X 0,Y 636.016,Z 1109.087,A -85,B 0,C 180,E1 27790.339,E2 27790.339} C_VEL
LIN {X 0,Y 637.265,Z 1092.109,A -85,B 0,C 180,E1 27788.913,E2 27788.913} C_VEL
LIN {X 0,Y 638.653,Z 1073.753,A -85,B 0,C 180,E1 27787.591,E2 27787.591} C_VEL
LIN {X 0,Y 640.023,Z 1055.415,A -85,B 0,C 180,E1 27786.465,E2 27786.465} C_VEL
LIN {X 0,Y 641.308,Z 1036.568,A -85,B 0,C 180,E1 27785.498,E2 27785.498} C_VEL
LIN {X 0,Y 642.602,Z 1015.712,A -85,B 0,C 180,E1 27784.617,E2 27784.617} C_VEL
LIN {X 0,Y 643.73,Z 995.056,A -85,B 0,C 180,E1 27783.918,E2 27783.918} C_VEL
LIN {X 0,Y 644.581,Z 974.555,A -85,B 0,C 180,E1 27783.394,E2 27783.394} C_VEL
LIN {X 0,Y 645.25,Z 951.87,A -85,B 0,C 180,E1 27782.989,E2 27782.989} C_VEL
LIN {X 0,Y 646.664,Z 814.901,A -85,B 0,C 180,E1 27781.375,E2 27781.375} C_VEL
LIN {X 0,Y 647.764,Z 670.742,A -85,B 0,C 180,E1 27779.695,E2 27779.695} C_VEL
LIN {X 0,Y 643.046,Z 644.507,A -85,B 0,C 180,E1 27779.064,E2 27779.064} C_VEL
LIN {X 0,Y 645.313,Z 596.794,A -85,B 0,C 180,E1 27775.883,E2 27775.883} C_VEL
LIN {X 0,Y 647.631,Z 553.535,A -85,B 0,C 180,E1 27772.924,E2 27772.924} C_VEL
LIN {X 0,Y 648.77,Z 533.557,A -85,B 0,C 180,E1 27771.53,E2 27771.53} C_VEL
LIN {X 0,Y 640.116,Z 511.82,A -85,B 0,C 180,E1 27769.238,E2 27769.238} C_VEL
LIN {X 0,Y 633.835,Z 497.297,A -85,B 0,C 180,E1 27767.586,E2 27767.586} C_VEL
LIN {X 0,Y 632.883,Z 494.563,A -85,B 0,C 180,E1 27767.242,E2 27767.242} C_VEL
LIN {X 0,Y 632.887,Z 494.382,A -85,B 0,C 180,E1 27764.292,E2 27764.292} C_VEL
LIN {X 0,Y 632.859,Z 494.391,A -85,B 0,C 180,E1 27761.212,E2 27761.212} C_VEL
LIN {X 0,Y 632.886,Z 494.357,A -85,B 0,C 180,E1 27758.151,E2 27758.151} C_VEL
LIN {X 0,Y 632.857,Z 494.397,A -85,B 0,C 180,E1 27754.997,E2 27754.997} C_VEL
LIN {X 0,Y 632.89,Z 494.399,A -85,B 0,C 180,E1 27751.956,E2 27751.956} C_VEL
LIN {X 0,Y 632.861,Z 494.394,A -85,B 0,C 180,E1 27748.912,E2 27748.912} C_VEL
LIN {X 0,Y 632.89,Z 494.391,A -85,B 0,C 180,E1 27745.852,E2 27745.852} C_VEL
LIN {X 0,Y 632.855,Z 494.383,A -85,B 0,C 180,E1 27742.676,E2 27742.676} C_VEL
LIN {X 0,Y 632.89,Z 494.386,A -85,B 0,C 180,E1 27739.665,E2 27739.665} C_VEL
LIN {X 0,Y 632.856,Z 494.394,A -85,B 0,C 180,E1 27736.523,E2 27736.523} C_VEL
LIN {X 0,Y 632.889,Z 494.391,A -85,B 0,C 180,E1 27733.522,E2 27733.522} C_VEL
LIN {X 0,Y 632.855,Z 494.381,A -85,B 0,C 180,E1 27730.377,E2 27730.377} C_VEL
LIN {X 0,Y 632.89,Z 494.394,A -85,B 0,C 180,E1 27727.352,E2 27727.352} C_VEL
LIN {X 0,Y 632.852,Z 494.393,A -85,B 0,C 180,E1 27724.168,E2 27724.168} C_VEL
LIN {X 0,Y 632.891,Z 494.384,A -85,B 0,C 180,E1 27721.086,E2 27721.086} C_VEL
LIN {X 0,Y 632.853,Z 494.393,A -85,B 0,C 180,E1 27718.008,E2 27718.008} C_VEL
LIN {X 0,Y 632.888,Z 494.394,A -85,B 0,C 180,E1 27714.924,E2 27714.924} C_VEL
LIN {X 0,Y 632.849,Z 494.38,A -85,B 0,C 180,E1 27711.825,E2 27711.825} C_VEL
LIN {X 0,Y 632.886,Z 494.393,A -85,B 0,C 180,E1 27708.795,E2 27708.795} C_VEL
LIN {X 0,Y 632.849,Z 494.394,A -85,B 0,C 180,E1 27705.637,E2 27705.637} C_VEL
LIN {X 0,Y 632.885,Z 494.386,A -85,B 0,C 180,E1 27702.596,E2 27702.596} C_VEL
LIN {X 0,Y 632.847,Z 494.387,A -85,B 0,C 180,E1 27699.466,E2 27699.466} C_VEL
LIN {X 0,Y 632.875,Z 494.398,A -85,B 0,C 180,E1 27696.538,E2 27696.538} C_VEL
LIN {X 0,Y 632.851,Z 494.396,A -85,B 0,C 180,E1 27693.339,E2 27693.339} C_VEL
LIN {X 0,Y 632.862,Z 494.394,A -85,B 0,C 180,E1 27690.466,E2 27690.466} C_VEL
LIN {X 0,Y 632.846,Z 494.361,A -85,B 0,C 180,E1 27687.196,E2 27687.196} C_VEL
LIN {X 0,Y 632.867,Z 494.396,A -85,B 0,C 180,E1 27684.227,E2 27684.227} C_VEL
LIN {X 0,Y 632.843,Z 494.358,A -85,B 0,C 180,E1 27681.017,E2 27681.017} C_VEL
LIN {X 0,Y 632.862,Z 494.396,A -85,B 0,C 180,E1 27678.084,E2 27678.084} C_VEL
LIN {X 0,Y 632.844,Z 494.384,A -85,B 0,C 180,E1 27674.812,E2 27674.812} C_VEL
LIN {X 0,Y 632.905,Z 494.607,A -85,B 0,C 180,E1 27673.072,E2 27673.072} C_VEL
LIN {X 0,Y 635.562,Z 501.172,A -85,B 0,C 180,E1 27672.317,E2 27672.317} C_VEL
LIN {X 0,Y 643.739,Z 519.872,A -85,B 0,C 180,E1 27670.301,E2 27670.301} C_VEL
LIN {X 0,Y 649.584,Z 534.351,A -85,B 0,C 180,E1 27668.877,E2 27668.877} C_VEL
LIN {X 0,Y 653.467,Z 554.621,A -85,B 0,C 180,E1 27668.351,E2 27668.351} C_VEL
LIN {X 0,Y 650.376,Z 785.596,A -85,B 0,C 180,E1 27665.455,E2 27665.455} C_VEL
LIN {X 0,Y 648.846,Z 921.175,A -85,B 0,C 180,E1 27663.793,E2 27663.793} C_VEL
LIN {X 0,Y 648.102,Z 946.487,A -85,B 0,C 180,E1 27663.327,E2 27663.327} C_VEL
LIN {X 0,Y 647.299,Z 967.951,A -85,B 0,C 180,E1 27662.799,E2 27662.799} C_VEL
LIN {X 0,Y 646.165,Z 993.226,A -85,B 0,C 180,E1 27662.006,E2 27662.006} C_VEL
LIN {X 0,Y 645.1,Z 1014.015,A -85,B 0,C 180,E1 27661.208,E2 27661.208} C_VEL
LIN {X 0,Y 643.668,Z 1038.458,A -85,B 0,C 180,E1 27660.087,E2 27660.087} C_VEL
LIN {X 0,Y 642.528,Z 1055.912,A -85,B 0,C 180,E1 27659.148,E2 27659.148} C_VEL
LIN {X 0,Y 640.999,Z 1076.143,A -85,B 0,C 180,E1 27657.869,E2 27657.869} C_VEL
LIN {X 0,Y 639.427,Z 1095.832,A -85,B 0,C 180,E1 27656.415,E2 27656.415} C_VEL
LIN {X 0,Y 637.985,Z 1114.177,A -85,B 0,C 180,E1 27654.885,E2 27654.885} C_VEL
LIN {X 0,Y 636.645,Z 1131.534,A -85,B 0,C 180,E1 27653.216,E2 27653.216} C_VEL
LIN {X 0,Y 635.554,Z 1146.513,A -85,B 0,C 180,E1 27651.596,E2 27651.596} C_VEL
LIN {X 0,Y 634.479,Z 1162.522,A -85,B 0,C 180,E1 27649.613,E2 27649.613} C_VEL
LIN {X 0,Y 633.675,Z 1175.79,A -85,B 0,C 180,E1 27647.73,E2 27647.73} C_VEL
LIN {X 0,Y 633.012,Z 1188.287,A -85,B 0,C 180,E1 27645.67,E2 27645.67} C_VEL
LIN {X 0,Y 632.586,Z 1198.021,A -85,B 0,C 180,E1 27643.808,E2 27643.808} C_VEL
LIN {X 0,Y 632.249,Z 1207.837,A -85,B 0,C 180,E1 27641.586,E2 27641.586} C_VEL
LIN {X 0,Y 632.072,Z 1214.818,A -85,B 0,C 180,E1 27639.653,E2 27639.653} C_VEL
LIN {X 0,Y 631.949,Z 1221.016,A -85,B 0,C 180,E1 27637.546,E2 27637.546} C_VEL
LIN {X 0,Y 631.905,Z 1225.496,A -85,B 0,C 180,E1 27635.448,E2 27635.448} C_VEL
LIN {X 0,Y 631.911,Z 1228.351,A -85,B 0,C 180,E1 27633.538,E2 27633.538} C_VEL
LIN {X 0,Y 631.907,Z 1230.191,A -85,B 0,C 180,E1 27631.269,E2 27631.269} C_VEL
LIN {X 0,Y 631.885,Z 1230.327,A -85,B 0,C 180,E1 27629.275,E2 27629.275} C_VEL
LIN {X 0,Y 631.886,Z 1229.224,A -85,B 0,C 180,E1 27627.279,E2 27627.279} C_VEL
LIN {X 0,Y 631.901,Z 1226.293,A -85,B 0,C 180,E1 27625.007,E2 27625.007} C_VEL
LIN {X 0,Y 631.954,Z 1222.69,A -85,B 0,C 180,E1 27623.185,E2 27623.185} C_VEL
LIN {X 0,Y 632.032,Z 1216.936,A -85,B 0,C 180,E1 27620.99,E2 27620.99} C_VEL
LIN {X 0,Y 632.188,Z 1209.604,A -85,B 0,C 180,E1 27618.875,E2 27618.875} C_VEL
LIN {X 0,Y 632.469,Z 1201.533,A -85,B 0,C 180,E1 27616.934,E2 27616.934} C_VEL
LIN {X 0,Y 632.902,Z 1190.865,A -85,B 0,C 180,E1 27614.797,E2 27614.797} C_VEL
LIN {X 0,Y 633.438,Z 1179.974,A -85,B 0,C 180,E1 27612.927,E2 27612.927} C_VEL
LIN {X 0,Y 634.275,Z 1165.474,A -85,B 0,C 180,E1 27610.784,E2 27610.784} C_VEL
LIN {X 0,Y 635.169,Z 1152.083,A -85,B 0,C 180,E1 27609.063,E2 27609.063} C_VEL
LIN {X 0,Y 636.44,Z 1134.312,A -85,B 0,C 180,E1 27607.07,E2 27607.07} C_VEL
LIN {X 0,Y 637.623,Z 1118.806,A -85,B 0,C 180,E1 27605.545,E2 27605.545} C_VEL
LIN {X 0,Y 639.182,Z 1098.871,A -85,B 0,C 180,E1 27603.824,E2 27603.824} C_VEL
LIN {X 0,Y 640.539,Z 1081.736,A -85,B 0,C 180,E1 27602.531,E2 27602.531} C_VEL
LIN {X 0,Y 642.171,Z 1060.799,A -85,B 0,C 180,E1 27601.14,E2 27601.14} C_VEL
LIN {X 0,Y 643.372,Z 1042.853,A -85,B 0,C 180,E1 27600.137,E2 27600.137} C_VEL
LIN {X 0,Y 644.602,Z 1022.879,A -85,B 0,C 180,E1 27599.174,E2 27599.174} C_VEL
LIN {X 0,Y 645.899,Z 998.93,A -85,B 0,C 180,E1 27598.2,E2 27598.2} C_VEL
LIN {X 0,Y 646.88,Z 977.897,A -85,B 0,C 180,E1 27597.492,E2 27597.492} C_VEL
LIN {X 0,Y 647.846,Z 953.018,A -85,B 0,C 180,E1 27596.817,E2 27596.817} C_VEL
LIN {X 0,Y 648.58,Z 930.623,A -85,B 0,C 180,E1 27596.363,E2 27596.363} C_VEL
LIN {X 0,Y 649.127,Z 904.031,A -85,B 0,C 180,E1 27595.979,E2 27595.979} C_VEL
LIN {X 0,Y 651.422,Z 696.344,A -85,B 0,C 180,E1 27593.447,E2 27593.447} C_VEL
LIN {X 0,Y 653.327,Z 552.932,A -85,B 0,C 180,E1 27591.618,E2 27591.618} C_VEL
LIN {X 0,Y 649.426,Z 533.993,A -85,B 0,C 180,E1 27591.105,E2 27591.105} C_VEL
LIN {X 0,Y 640.59,Z 512.58,A -85,B 0,C 180,E1 27588.931,E2 27588.931} C_VEL
LIN {X 0,Y 634.045,Z 497.705,A -85,B 0,C 180,E1 27587.298,E2 27587.298} C_VEL
LIN {X 0,Y 632.897,Z 494.531,A -85,B 0,C 180,E1 27586.901,E2 27586.901} C_VEL
LIN {X 0,Y 632.841,Z 494.364,A -85,B 0,C 180,E1 27583.777,E2 27583.777} C_VEL
LIN {X 0,Y 632.869,Z 494.393,A -85,B 0,C 180,E1 27580.821,E2 27580.821} C_VEL
LIN {X 0,Y 632.851,Z 494.379,A -85,B 0,C 180,E1 27577.67,E2 27577.67} C_VEL
LIN {X 0,Y 632.858,Z 494.38,A -85,B 0,C 180,E1 27574.76,E2 27574.76} C_VEL
LIN {X 0,Y 632.857,Z 494.384,A -85,B 0,C 180,E1 27571.532,E2 27571.532} C_VEL
LIN {X 0,Y 632.856,Z 494.388,A -85,B 0,C 180,E1 27568.603,E2 27568.603} C_VEL
LIN {X 0,Y 632.861,Z 494.388,A -85,B 0,C 180,E1 27565.351,E2 27565.351} C_VEL
LIN {X 0,Y 632.862,Z 494.394,A -85,B 0,C 180,E1 27562.381,E2 27562.381} C_VEL
LIN {X 0,Y 632.858,Z 494.399,A -85,B 0,C 180,E1 27559.09,E2 27559.09} C_VEL
LIN {X 0,Y 632.878,Z 494.385,A -85,B 0,C 180,E1 27556.051,E2 27556.051} C_VEL
LIN {X 0,Y 632.855,Z 494.386,A -85,B 0,C 180,E1 27552.872,E2 27552.872} C_VEL
LIN {X 0,Y 632.884,Z 494.392,A -85,B 0,C 180,E1 27549.824,E2 27549.824} C_VEL
LIN {X 0,Y 632.854,Z 494.397,A -85,B 0,C 180,E1 27546.623,E2 27546.623} C_VEL
LIN {X 0,Y 632.887,Z 494.38,A -85,B 0,C 180,E1 27543.533,E2 27543.533} C_VEL
LIN {X 0,Y 632.853,Z 494.392,A -85,B 0,C 180,E1 27540.362,E2 27540.362} C_VEL
LIN {X 0,Y 632.89,Z 494.388,A -85,B 0,C 180,E1 27537.283,E2 27537.283} C_VEL
LIN {X 0,Y 632.855,Z 494.386,A -85,B 0,C 180,E1 27534.196,E2 27534.196} C_VEL
LIN {X 0,Y 632.892,Z 494.391,A -85,B 0,C 180,E1 27531.185,E2 27531.185} C_VEL
LIN {X 0,Y 632.86,Z 494.399,A -85,B 0,C 180,E1 27528.055,E2 27528.055} C_VEL
LIN {X 0,Y 632.893,Z 494.378,A -85,B 0,C 180,E1 27524.983,E2 27524.983} C_VEL
LIN {X 0,Y 632.861,Z 494.388,A -85,B 0,C 180,E1 27521.865,E2 27521.865} C_VEL
LIN {X 0,Y 632.892,Z 494.392,A -85,B 0,C 180,E1 27518.763,E2 27518.763} C_VEL
LIN {X 0,Y 632.861,Z 494.399,A -85,B 0,C 180,E1 27515.646,E2 27515.646} C_VEL
LIN {X 0,Y 632.888,Z 494.385,A -85,B 0,C 180,E1 27512.527,E2 27512.527} C_VEL
LIN {X 0,Y 632.862,Z 494.393,A -85,B 0,C 180,E1 27509.42,E2 27509.42} C_VEL
LIN {X 0,Y 632.886,Z 494.385,A -85,B 0,C 180,E1 27506.321,E2 27506.321} C_VEL
LIN {X 0,Y 632.859,Z 494.372,A -85,B 0,C 180,E1 27503.215,E2 27503.215} C_VEL
LIN {X 0,Y 632.885,Z 494.391,A -85,B 0,C 180,E1 27500.101,E2 27500.101} C_VEL
LIN {X 0,Y 632.861,Z 494.361,A -85,B 0,C 180,E1 27497.012,E2 27497.012} C_VEL
LIN {X 0,Y 632.886,Z 494.375,A -85,B 0,C 180,E1 27494.037,E2 27494.037} C_VEL
LIN {X 0,Y 632.898,Z 494.621,A -85,B 0,C 180,E1 27492.649,E2 27492.649} C_VEL
LIN {X 0,Y 633.832,Z 497.267,A -85,B 0,C 180,E1 27492.321,E2 27492.321} C_VEL
LIN {X 0,Y 635.13,Z 501.506,A -85,B 0,C 180,E1 27491.875,E2 27491.875} C_VEL
LIN {X 0,Y 635.244,Z 509.858,A -85,B 0,C 180,E1 27491.203,E2 27491.203} C_VEL
LIN {X 0,Y 635.236,Z 518.363,A -85,B 0,C 180,E1 27490.536,E2 27490.536} C_VEL
LIN {X 0,Y 636.378,Z 522.844,A -85,B 0,C 180,E1 27490.099,E2 27490.099} C_VEL
LIN {X 0,Y 641.908,Z 537.221,A -85,B 0,C 180,E1 27488.591,E2 27488.591} C_VEL
LIN {X 0,Y 639.095,Z 584.185,A -85,B 0,C 180,E1 27485.315,E2 27485.315} C_VEL
LIN {X 0,Y 636.661,Z 629.717,A -85,B 0,C 180,E1 27482.22,E2 27482.22} C_VEL
LIN {X 0,Y 636.034,Z 644.493,A -85,B 0,C 180,E1 27481.256,E2 27481.256} C_VEL
LIN {X 0,Y 641.269,Z 674.18,A -85,B 0,C 180,E1 27480.561,E2 27480.561} C_VEL
LIN {X 0,Y 638.84,Z 937.263,A -85,B 0,C 180,E1 27477.505,E2 27477.505} C_VEL
LIN {X 0,Y 638.299,Z 963.003,A -85,B 0,C 180,E1 27477.144,E2 27477.144} C_VEL
LIN {X 0,Y 637.52,Z 984.131,A -85,B 0,C 180,E1 27476.695,E2 27476.695} C_VEL
LIN {X 0,Y 636.494,Z 1004.381,A -85,B 0,C 180,E1 27476.094,E2 27476.094} C_VEL
LIN {X 0,Y 635.183,Z 1025.424,A -85,B 0,C 180,E1 27475.301,E2 27475.301} C_VEL
LIN {X 0,Y 633.778,Z 1045.511,A -85,B 0,C 180,E1 27474.365,E2 27474.365} C_VEL
LIN {X 0,Y 632.26,Z 1064.446,A -85,B 0,C 180,E1 27473.288,E2 27473.288} C_VEL
LIN {X 0,Y 630.734,Z 1083.018,A -85,B 0,C 180,E1 27472.042,E2 27472.042} C_VEL
LIN {X 0,Y 629.331,Z 1100.14,A -85,B 0,C 180,E1 27470.701,E2 27470.701} C_VEL
LIN {X 0,Y 627.995,Z 1116.515,A -85,B 0,C 180,E1 27469.195,E2 27469.195} C_VEL
LIN {X 0,Y 626.817,Z 1131.89,A -85,B 0,C 180,E1 27467.546,E2 27467.546} C_VEL
LIN {X 0,Y 625.892,Z 1145.561,A -85,B 0,C 180,E1 27465.853,E2 27465.853} C_VEL
LIN {X 0,Y 625.158,Z 1157.857,A -85,B 0,C 180,E1 27464.07,E2 27464.07} C_VEL
LIN {X 0,Y 624.618,Z 1168.718,A -85,B 0,C 180,E1 27462.198,E2 27462.198} C_VEL
LIN {X 0,Y 624.258,Z 1178.684,A -85,B 0,C 180,E1 27460.148,E2 27460.148} C_VEL
LIN {X 0,Y 624.074,Z 1186.405,A -85,B 0,C 180,E1 27458.198,E2 27458.198} C_VEL
LIN {X 0,Y 623.964,Z 1192.295,A -85,B 0,C 180,E1 27456.256,E2 27456.256} C_VEL
LIN {X 0,Y 623.928,Z 1196.702,A -85,B 0,C 180,E1 27454.227,E2 27454.227} C_VEL
LIN {X 0,Y 623.914,Z 1199.369,A -85,B 0,C 180,E1 27452.296,E2 27452.296} C_VEL
LIN {X 0,Y 623.903,Z 1200.401,A -85,B 0,C 180,E1 27450.367,E2 27450.367} C_VEL
LIN {X 0,Y 623.911,Z 1199.847,A -85,B 0,C 180,E1 27448.255,E2 27448.255} C_VEL
LIN {X 0,Y 623.918,Z 1197.81,A -85,B 0,C 180,E1 27446.325,E2 27446.325} C_VEL
LIN {X 0,Y 623.942,Z 1194.049,A -85,B 0,C 180,E1 27444.373,E2 27444.373} C_VEL
LIN {X 0,Y 624.016,Z 1188.518,A -85,B 0,C 180,E1 27442.358,E2 27442.358} C_VEL
LIN {X 0,Y 624.188,Z 1181.506,A -85,B 0,C 180,E1 27440.41,E2 27440.41} C_VEL
LIN {X 0,Y 624.465,Z 1172.55,A -85,B 0,C 180,E1 27438.455,E2 27438.455} C_VEL
LIN {X 0,Y 624.922,Z 1162.374,A -85,B 0,C 180,E1 27436.585,E2 27436.585} C_VEL
LIN {X 0,Y 625.558,Z 1150.965,A -85,B 0,C 180,E1 27434.804,E2 27434.804} C_VEL
LIN {X 0,Y 626.37,Z 1138.187,A -85,B 0,C 180,E1 27433.111,E2 27433.111} C_VEL
LIN {X 0,Y 627.453,Z 1123.316,A -85,B 0,C 180,E1 27431.416,E2 27431.416} C_VEL
LIN {X 0,Y 628.722,Z 1107.518,A -85,B 0,C 180,E1 27429.861,E2 27429.861} C_VEL
LIN {X 0,Y 630.047,Z 1091.357,A -85,B 0,C 180,E1 27428.495,E2 27428.495} C_VEL
LIN {X 0,Y 631.499,Z 1073.802,A -85,B 0,C 180,E1 27427.225,E2 27427.225} C_VEL
LIN {X 0,Y 633.038,Z 1054.832,A -85,B 0,C 180,E1 27426.051,E2 27426.051} C_VEL
LIN {X 0,Y 634.485,Z 1035.758,A -85,B 0,C 180,E1 27425.068,E2 27425.068} C_VEL
LIN {X 0,Y 635.797,Z 1015.903,A -85,B 0,C 180,E1 27424.226,E2 27424.226} C_VEL
LIN {X 0,Y 637.013,Z 995.04,A -85,B 0,C 180,E1 27423.517,E2 27423.517} C_VEL
LIN {X 0,Y 637.896,Z 974.791,A -85,B 0,C 180,E1 27422.998,E2 27422.998} C_VEL
LIN {X 0,Y 638.601,Z 951.953,A -85,B 0,C 180,E1 27422.589,E2 27422.589} C_VEL
LIN {X 0,Y 640.302,Z 776.526,A -85,B 0,C 180,E1 27420.537,E2 27420.537} C_VEL
LIN {X 0,Y 641.103,Z 672.051,A -85,B 0,C 180,E1 27419.311,E2 27419.311} C_VEL
LIN {X 0,Y 635.984,Z 643.634,A -85,B 0,C 180,E1 27418.617,E2 27418.617} C_VEL
LIN {X 0,Y 638.555,Z 593.801,A -85,B 0,C 180,E1 27415.253,E2 27415.253} C_VEL
LIN {X 0,Y 641.143,Z 549.776,A -85,B 0,C 180,E1 27412.202,E2 27412.202} C_VEL
LIN {X 0,Y 641.903,Z 536.993,A -85,B 0,C 180,E1 27411.298,E2 27411.298} C_VEL
LIN {X 0,Y 633.527,Z 515.924,A -85,B 0,C 180,E1 27409.044,E2 27409.044} C_VEL
LIN {X 0,Y 626.41,Z 499.143,A -85,B 0,C 180,E1 27407.111,E2 27407.111} C_VEL
LIN {X 0,Y 624.966,Z 495.55,A -85,B 0,C 180,E1 27406.649,E2 27406.649} C_VEL
LIN {X 0,Y 624.926,Z 495.351,A -85,B 0,C 180,E1 27403.416,E2 27403.416} C_VEL
LIN {X 0,Y 624.955,Z 495.386,A -85,B 0,C 180,E1 27400.258,E2 27400.258} C_VEL
LIN {X 0,Y 624.918,Z 495.352,A -85,B 0,C 180,E1 27397.101,E2 27397.101} C_VEL
LIN {X 0,Y 624.951,Z 495.378,A -85,B 0,C 180,E1 27394.03,E2 27394.03} C_VEL
LIN {X 0,Y 624.92,Z 495.383,A -85,B 0,C 180,E1 27390.905,E2 27390.905} C_VEL
LIN {X 0,Y 624.954,Z 495.38,A -85,B 0,C 180,E1 27387.852,E2 27387.852} C_VEL
LIN {X 0,Y 624.915,Z 495.385,A -85,B 0,C 180,E1 27384.661,E2 27384.661} C_VEL
LIN {X 0,Y 624.954,Z 495.385,A -85,B 0,C 180,E1 27381.592,E2 27381.592} C_VEL
LIN {X 0,Y 624.914,Z 495.373,A -85,B 0,C 180,E1 27378.47,E2 27378.47} C_VEL
LIN {X 0,Y 624.952,Z 495.371,A -85,B 0,C 180,E1 27375.402,E2 27375.402} C_VEL
LIN {X 0,Y 624.912,Z 495.385,A -85,B 0,C 180,E1 27372.287,E2 27372.287} C_VEL
LIN {X 0,Y 624.952,Z 495.38,A -85,B 0,C 180,E1 27369.201,E2 27369.201} C_VEL
LIN {X 0,Y 624.911,Z 495.375,A -85,B 0,C 180,E1 27366.154,E2 27366.154} C_VEL
LIN {X 0,Y 624.951,Z 495.384,A -85,B 0,C 180,E1 27363.118,E2 27363.118} C_VEL
LIN {X 0,Y 624.91,Z 495.379,A -85,B 0,C 180,E1 27359.959,E2 27359.959} C_VEL
LIN {X 0,Y 624.952,Z 495.371,A -85,B 0,C 180,E1 27356.882,E2 27356.882} C_VEL
LIN {X 0,Y 624.908,Z 495.385,A -85,B 0,C 180,E1 27353.754,E2 27353.754} C_VEL
LIN {X 0,Y 624.953,Z 495.379,A -85,B 0,C 180,E1 27350.7,E2 27350.7} C_VEL
LIN {X 0,Y 624.906,Z 495.374,A -85,B 0,C 180,E1 27347.619,E2 27347.619} C_VEL
LIN {X 0,Y 624.956,Z 495.381,A -85,B 0,C 180,E1 27344.598,E2 27344.598} C_VEL
LIN {X 0,Y 624.907,Z 495.384,A -85,B 0,C 180,E1 27341.433,E2 27341.433} C_VEL
LIN {X 0,Y 624.954,Z 495.375,A -85,B 0,C 180,E1 27338.362,E2 27338.362} C_VEL
LIN {X 0,Y 624.903,Z 495.375,A -85,B 0,C 180,E1 27335.215,E2 27335.215} C_VEL
LIN {X 0,Y 624.954,Z 495.375,A -85,B 0,C 180,E1 27332.148,E2 27332.148} C_VEL
LIN {X 0,Y 624.904,Z 495.385,A -85,B 0,C 180,E1 27329.049,E2 27329.049} C_VEL
LIN {X 0,Y 624.948,Z 495.345,A -85,B 0,C 180,E1 27325.97,E2 27325.97} C_VEL
LIN {X 0,Y 624.901,Z 495.387,A -85,B 0,C 180,E1 27322.898,E2 27322.898} C_VEL
LIN {X 0,Y 624.951,Z 495.354,A -85,B 0,C 180,E1 27319.851,E2 27319.851} C_VEL
LIN {X 0,Y 624.897,Z 495.354,A -85,B 0,C 180,E1 27316.72,E2 27316.72} C_VEL
LIN {X 0,Y 624.959,Z 495.485,A -85,B 0,C 180,E1 27313.721,E2 27313.721} C_VEL
LIN {X 0,Y 625.276,Z 496.823,A -85,B 0,C 180,E1 27313.514,E2 27313.514} C_VEL
LIN {X 0,Y 633.257,Z 514.824,A -85,B 0,C 180,E1 27311.477,E2 27311.477} C_VEL
LIN {X 0,Y 641.166,Z 534.003,A -85,B 0,C 180,E1 27309.471,E2 27309.471} C_VEL
LIN {X 0,Y 642.619,Z 536.881,A -85,B 0,C 180,E1 27309.277,E2 27309.277} C_VEL
LIN {X 0,Y 643.65,Z 539.168,A -85,B 0,C 180,E1 27309.178,E2 27309.178} C_VEL
LIN {X 0,Y 646.863,Z 556.275,A -85,B 0,C 180,E1 27308.734,E2 27308.734} C_VEL
LIN {X 0,Y 643.364,Z 791.431,A -85,B 0,C 180,E1 27305.738,E2 27305.738} C_VEL
LIN {X 0,Y 641.724,Z 922.104,A -85,B 0,C 180,E1 27304.108,E2 27304.108} C_VEL
LIN {X 0,Y 640.94,Z 946.929,A -85,B 0,C 180,E1 27303.641,E2 27303.641} C_VEL
LIN {X 0,Y 640.119,Z 967.753,A -85,B 0,C 180,E1 27303.124,E2 27303.124} C_VEL
LIN {X 0,Y 638.904,Z 993.258,A -85,B 0,C 180,E1 27302.316,E2 27302.316} C_VEL
LIN {X 0,Y 637.764,Z 1014.142,A -85,B 0,C 180,E1 27301.506,E2 27301.506} C_VEL
LIN {X 0,Y 636.294,Z 1038.095,A -85,B 0,C 180,E1 27300.397,E2 27300.397} C_VEL
LIN {X 0,Y 634.977,Z 1057.371,A -85,B 0,C 180,E1 27299.35,E2 27299.35} C_VEL
LIN {X 0,Y 633.446,Z 1078.826,A -85,B 0,C 180,E1 27298.007,E2 27298.007} C_VEL
LIN {X 0,Y 632.181,Z 1094.324,A -85,B 0,C 180,E1 27296.867,E2 27296.867} C_VEL
LIN {X 0,Y 630.789,Z 1110.849,A -85,B 0,C 180,E1 27295.49,E2 27295.49} C_VEL
LIN {X 0,Y 629.213,Z 1129.681,A -85,B 0,C 180,E1 27293.705,E2 27293.705} C_VEL
LIN {X 0,Y 628.012,Z 1144.785,A -85,B 0,C 180,E1 27292.07,E2 27292.07} C_VEL
LIN {X 0,Y 626.82,Z 1161.119,A -85,B 0,C 180,E1 27290.057,E2 27290.057} C_VEL
LIN {X 0,Y 625.949,Z 1173.883,A -85,B 0,C 180,E1 27288.245,E2 27288.245} C_VEL
LIN {X 0,Y 625.211,Z 1186.735,A -85,B 0,C 180,E1 27286.157,E2 27286.157} C_VEL
LIN {X 0,Y 624.699,Z 1197.103,A -85,B 0,C 180,E1 27284.175,E2 27284.175} C_VEL
LIN {X 0,Y 624.335,Z 1206.772,A -85,B 0,C 180,E1 27282.016,E2 27282.016} C_VEL
LIN {X 0,Y 624.091,Z 1214.212,A -85,B 0,C 180,E1 27279.964,E2 27279.964} C_VEL
LIN {X 0,Y 623.985,Z 1220,A -85,B 0,C 180,E1 27278.013,E2 27278.013} C_VEL
LIN {X 0,Y 623.925,Z 1225.176,A -85,B 0,C 180,E1 27275.702,E2 27275.702} C_VEL
LIN {X 0,Y 623.913,Z 1228.124,A -85,B 0,C 180,E1 27273.767,E2 27273.767} C_VEL
LIN {X 0,Y 623.897,Z 1230.103,A -85,B 0,C 180,E1 27271.561,E2 27271.561} C_VEL
LIN {X 0,Y 623.884,Z 1230.373,A -85,B 0,C 180,E1 27269.449,E2 27269.449} C_VEL
LIN {X 0,Y 623.899,Z 1229.428,A -85,B 0,C 180,E1 27267.52,E2 27267.52} C_VEL
LIN {X 0,Y 623.912,Z 1226.769,A -85,B 0,C 180,E1 27265.22,E2 27265.22} C_VEL
LIN {X 0,Y 623.956,Z 1222.896,A -85,B 0,C 180,E1 27263.19,E2 27263.19} C_VEL
LIN {X 0,Y 624.027,Z 1217.711,A -85,B 0,C 180,E1 27261.152,E2 27261.152} C_VEL
LIN {X 0,Y 624.2,Z 1210.309,A -85,B 0,C 180,E1 27258.918,E2 27258.918} C_VEL
LIN {X 0,Y 624.491,Z 1202.347,A -85,B 0,C 180,E1 27256.953,E2 27256.953} C_VEL
LIN {X 0,Y 624.974,Z 1191.378,A -85,B 0,C 180,E1 27254.694,E2 27254.694} C_VEL
LIN {X 0,Y 625.548,Z 1180.546,A -85,B 0,C 180,E1 27252.801,E2 27252.801} C_VEL
LIN {X 0,Y 626.415,Z 1166.724,A -85,B 0,C 180,E1 27250.707,E2 27250.707} C_VEL
LIN {X 0,Y 627.346,Z 1153.622,A -85,B 0,C 180,E1 27248.986,E2 27248.986} C_VEL
LIN {X 0,Y 628.564,Z 1138.007,A -85,B 0,C 180,E1 27247.162,E2 27247.162} C_VEL
LIN {X 0,Y 629.943,Z 1120.832,A -85,B 0,C 180,E1 27245.427,E2 27245.427} C_VEL
LIN {X 0,Y 631.501,Z 1102.509,A -85,B 0,C 180,E1 27243.785,E2 27243.785} C_VEL
LIN {X 0,Y 633.007,Z 1084.538,A -85,B 0,C 180,E1 27242.394,E2 27242.394} C_VEL
LIN {X 0,Y 634.267,Z 1067.528,A -85,B 0,C 180,E1 27241.262,E2 27241.262} C_VEL
LIN {X 0,Y 635.779,Z 1045.661,A -85,B 0,C 180,E1 27239.993,E2 27239.993} C_VEL
LIN {X 0,Y 637.11,Z 1024.967,A -85,B 0,C 180,E1 27238.971,E2 27238.971} C_VEL
LIN {X 0,Y 638.494,Z 1001.65,A -85,B 0,C 180,E1 27237.989,E2 27237.989} C_VEL
LIN {X 0,Y 639.587,Z 979.559,A -85,B 0,C 180,E1 27237.227,E2 27237.227} C_VEL
LIN {X 0,Y 640.608,Z 955.971,A -85,B 0,C 180,E1 27236.56,E2 27236.56} C_VEL
LIN {X 0,Y 641.416,Z 931.857,A -85,B 0,C 180,E1 27236.058,E2 27236.058} C_VEL
LIN {X 0,Y 642.01,Z 906.675,A -85,B 0,C 180,E1 27235.679,E2 27235.679} C_VEL
LIN {X 0,Y 644.146,Z 732.694,A -85,B 0,C 180,E1 27233.532,E2 27233.532} C_VEL
LIN {X 0,Y 646.762,Z 554.655,A -85,B 0,C 180,E1 27231.237,E2 27231.237} C_VEL
LIN {X 0,Y 643.158,Z 537.725,A -85,B 0,C 180,E1 27230.77,E2 27230.77} C_VEL
LIN {X 0,Y 641.377,Z 534.537,A -85,B 0,C 180,E1 27230.577,E2 27230.577} C_VEL
LIN {X 0,Y 633.808,Z 516.203,A -85,B 0,C 180,E1 27228.672,E2 27228.672} C_VEL
LIN {X 0,Y 626.228,Z 498.809,A -85,B 0,C 180,E1 27226.727,E2 27226.727} C_VEL
LIN {X 0,Y 624.972,Z 495.553,A -85,B 0,C 180,E1 27226.316,E2 27226.316} C_VEL
LIN {X 0,Y 624.895,Z 495.354,A -85,B 0,C 180,E1 27223.349,E2 27223.349} C_VEL
LIN {X 0,Y 624.955,Z 495.357,A -85,B 0,C 180,E1 27220.258,E2 27220.258} C_VEL
LIN {X 0,Y 624.899,Z 495.384,A -85,B 0,C 180,E1 27217.217,E2 27217.217} C_VEL
LIN {X 0,Y 624.949,Z 495.346,A -85,B 0,C 180,E1 27214.166,E2 27214.166} C_VEL
LIN {X 0,Y 624.903,Z 495.386,A -85,B 0,C 180,E1 27211.12,E2 27211.12} C_VEL
LIN {X 0,Y 624.955,Z 495.373,A -85,B 0,C 180,E1 27208.059,E2 27208.059} C_VEL
LIN {X 0,Y 624.903,Z 495.376,A -85,B 0,C 180,E1 27204.988,E2 27204.988} C_VEL
LIN {X 0,Y 624.96,Z 495.382,A -85,B 0,C 180,E1 27201.986,E2 27201.986} C_VEL
LIN {X 0,Y 624.907,Z 495.386,A -85,B 0,C 180,E1 27198.857,E2 27198.857} C_VEL
LIN {X 0,Y 624.953,Z 495.375,A -85,B 0,C 180,E1 27195.783,E2 27195.783} C_VEL
LIN {X 0,Y 624.907,Z 495.374,A -85,B 0,C 180,E1 27192.663,E2 27192.663} C_VEL
LIN {X 0,Y 624.953,Z 495.382,A -85,B 0,C 180,E1 27189.578,E2 27189.578} C_VEL
LIN {X 0,Y 624.91,Z 495.385,A -85,B 0,C 180,E1 27186.486,E2 27186.486} C_VEL
LIN {X 0,Y 624.95,Z 495.368,A -85,B 0,C 180,E1 27183.394,E2 27183.394} C_VEL
LIN {X 0,Y 624.912,Z 495.38,A -85,B 0,C 180,E1 27180.275,E2 27180.275} C_VEL
LIN {X 0,Y 624.951,Z 495.379,A -85,B 0,C 180,E1 27177.157,E2 27177.157} C_VEL
LIN {X 0,Y 624.913,Z 495.375,A -85,B 0,C 180,E1 27174.03,E2 27174.03} C_VEL
LIN {X 0,Y 624.951,Z 495.383,A -85,B 0,C 180,E1 27170.979,E2 27170.979} C_VEL
LIN {X 0,Y 624.916,Z 495.386,A -85,B 0,C 180,E1 27167.847,E2 27167.847} C_VEL
LIN {X 0,Y 624.948,Z 495.369,A -85,B 0,C 180,E1 27164.74,E2 27164.74} C_VEL
LIN {X 0,Y 624.916,Z 495.374,A -85,B 0,C 180,E1 27161.627,E2 27161.627} C_VEL
LIN {X 0,Y 624.949,Z 495.385,A -85,B 0,C 180,E1 27158.507,E2 27158.507} C_VEL
LIN {X 0,Y 624.918,Z 495.386,A -85,B 0,C 180,E1 27155.417,E2 27155.417} C_VEL
LIN {X 0,Y 624.948,Z 495.376,A -85,B 0,C 180,E1 27152.355,E2 27152.355} C_VEL
LIN {X 0,Y 624.921,Z 495.382,A -85,B 0,C 180,E1 27149.309,E2 27149.309} C_VEL
LIN {X 0,Y 624.946,Z 495.374,A -85,B 0,C 180,E1 27146.276,E2 27146.276} C_VEL
LIN {X 0,Y 624.922,Z 495.36,A -85,B 0,C 180,E1 27143.244,E2 27143.244} C_VEL
LIN {X 0,Y 624.949,Z 495.379,A -85,B 0,C 180,E1 27140.17,E2 27140.17} C_VEL
LIN {X 0,Y 624.922,Z 495.348,A -85,B 0,C 180,E1 27137.03,E2 27137.03} C_VEL
LIN {X 0,Y 624.944,Z 495.359,A -85,B 0,C 180,E1 27133.946,E2 27133.946} C_VEL
LIN {X 0,Y 624.974,Z 495.596,A -85,B 0,C 180,E1 27133.247,E2 27133.247} C_VEL
LIN {X 0,Y 627.549,Z 501.993,A -85,B 0,C 180,E1 27132.463,E2 27132.463} C_VEL
LIN {X 0,Y 635.742,Z 521.262,A -85,B 0,C 180,E1 27130.27,E2 27130.27} C_VEL
LIN {X 0,Y 636.378,Z 522.844,A -85,B 0,C 180,E1 27130.099,E2 27130.099} C_VEL
LIN {X 0,Y 637.139,Z 526.957,A -85,B 0,C 180,E1 27129.723,E2 27129.723} C_VEL
LIN {X 0,Y 636.193,Z 534.187,A -85,B 0,C 180,E1 27129.238,E2 27129.238} C_VEL
LIN {X 0,Y 634.976,Z 541.631,A -85,B 0,C 180,E1 27128.759,E2 27128.759} C_VEL
LIN {X 0,Y 632.023,Z 588.035,A -85,B 0,C 180,E1 27125.492,E2 27125.492} C_VEL
LIN {X 0,Y 629.372,Z 634.463,A -85,B 0,C 180,E1 27122.307,E2 27122.307} C_VEL
LIN {X 0,Y 629.027,Z 643.767,A -85,B 0,C 180,E1 27121.709,E2 27121.709} C_VEL
LIN {X 0,Y 634.637,Z 675.439,A -85,B 0,C 180,E1 27120.952,E2 27120.952} C_VEL
LIN {X 0,Y 632.032,Z 947.706,A -85,B 0,C 180,E1 27117.781,E2 27117.781} C_VEL
LIN {X 0,Y 631.443,Z 969.155,A -85,B 0,C 180,E1 27117.438,E2 27117.438} C_VEL
LIN {X 0,Y 630.534,Z 990.187,A -85,B 0,C 180,E1 27116.935,E2 27116.935} C_VEL
LIN {X 0,Y 629.439,Z 1010.111,A -85,B 0,C 180,E1 27116.307,E2 27116.307} C_VEL
LIN {X 0,Y 628.06,Z 1029.905,A -85,B 0,C 180,E1 27115.512,E2 27115.512} C_VEL
LIN {X 0,Y 626.475,Z 1050.053,A -85,B 0,C 180,E1 27114.517,E2 27114.517} C_VEL
LIN {X 0,Y 624.913,Z 1068.506,A -85,B 0,C 180,E1 27113.428,E2 27113.428} C_VEL
LIN {X 0,Y 623.248,Z 1086.667,A -85,B 0,C 180,E1 27112.148,E2 27112.148} C_VEL
LIN {X 0,Y 621.615,Z 1104.367,A -85,B 0,C 180,E1 27110.683,E2 27110.683} C_VEL
LIN {X 0,Y 620.202,Z 1120.484,A -85,B 0,C 180,E1 27109.134,E2 27109.134} C_VEL
LIN {X 0,Y 618.992,Z 1135.18,A -85,B 0,C 180,E1 27107.484,E2 27107.484} C_VEL
LIN {X 0,Y 617.998,Z 1148.248,A -85,B 0,C 180,E1 27105.772,E2 27105.772} C_VEL
LIN {X 0,Y 617.191,Z 1160.69,A -85,B 0,C 180,E1 27103.872,E2 27103.872} C_VEL
LIN {X 0,Y 616.649,Z 1171.185,A -85,B 0,C 180,E1 27101.978,E2 27101.978} C_VEL
LIN {X 0,Y 616.275,Z 1180.214,A -85,B 0,C 180,E1 27099.987,E2 27099.987} C_VEL
LIN {X 0,Y 616.05,Z 1187.711,A -85,B 0,C 180,E1 27097.93,E2 27097.93} C_VEL
LIN {X 0,Y 615.948,Z 1193.264,A -85,B 0,C 180,E1 27095.963,E2 27095.963} C_VEL
LIN {X 0,Y 615.923,Z 1197.182,A -85,B 0,C 180,E1 27094.003,E2 27094.003} C_VEL
LIN {X 0,Y 615.917,Z 1199.641,A -85,B 0,C 180,E1 27091.954,E2 27091.954} C_VEL
LIN {X 0,Y 615.913,Z 1200.491,A -85,B 0,C 180,E1 27089.907,E2 27089.907} C_VEL
LIN {X 0,Y 615.914,Z 1199.574,A -85,B 0,C 180,E1 27087.86,E2 27087.86} C_VEL
LIN {X 0,Y 615.925,Z 1197.016,A -85,B 0,C 180,E1 27085.811,E2 27085.811} C_VEL
LIN {X 0,Y 615.96,Z 1193.043,A -85,B 0,C 180,E1 27083.85,E2 27083.85} C_VEL
LIN {X 0,Y 616.06,Z 1187.396,A -85,B 0,C 180,E1 27081.883,E2 27081.883} C_VEL
LIN {X 0,Y 616.288,Z 1179.748,A -85,B 0,C 180,E1 27079.814,E2 27079.814} C_VEL
LIN {X 0,Y 616.654,Z 1170.978,A -85,B 0,C 180,E1 27077.892,E2 27077.892} C_VEL
LIN {X 0,Y 617.226,Z 1160.093,A -85,B 0,C 180,E1 27075.937,E2 27075.937} C_VEL
LIN {X 0,Y 618.001,Z 1148.198,A -85,B 0,C 180,E1 27074.132,E2 27074.132} C_VEL
LIN {X 0,Y 619.027,Z 1134.666,A -85,B 0,C 180,E1 27072.366,E2 27072.366} C_VEL
LIN {X 0,Y 620.269,Z 1119.802,A -85,B 0,C 180,E1 27070.704,E2 27070.704} C_VEL
LIN {X 0,Y 621.662,Z 1103.84,A -85,B 0,C 180,E1 27069.179,E2 27069.179} C_VEL
LIN {X 0,Y 623.336,Z 1085.624,A -85,B 0,C 180,E1 27067.684,E2 27067.684} C_VEL
LIN {X 0,Y 624.991,Z 1067.631,A -85,B 0,C 180,E1 27066.425,E2 27066.425} C_VEL
LIN {X 0,Y 626.569,Z 1049.016,A -85,B 0,C 180,E1 27065.336,E2 27065.336} C_VEL
LIN {X 0,Y 628.145,Z 1028.681,A -85,B 0,C 180,E1 27064.345,E2 27064.345} C_VEL
LIN {X 0,Y 629.559,Z 1008.53,A -85,B 0,C 180,E1 27063.546,E2 27063.546} C_VEL
LIN {X 0,Y 630.636,Z 988.095,A -85,B 0,C 180,E1 27062.917,E2 27062.917} C_VEL
LIN {X 0,Y 631.558,Z 965.462,A -85,B 0,C 180,E1 27062.405,E2 27062.405} C_VEL
LIN {X 0,Y 632.124,Z 943.233,A -85,B 0,C 180,E1 27062.072,E2 27062.072} C_VEL
LIN {X 0,Y 634.606,Z 674.181,A -85,B 0,C 180,E1 27058.938,E2 27058.938} C_VEL
LIN {X 0,Y 628.956,Z 642.72,A -85,B 0,C 180,E1 27058.158,E2 27058.158} C_VEL
LIN {X 0,Y 631.676,Z 593.845,A -85,B 0,C 180,E1 27054.819,E2 27054.819} C_VEL
LIN {X 0,Y 634.478,Z 549.417,A -85,B 0,C 180,E1 27051.704,E2 27051.704} C_VEL
LIN {X 0,Y 635.05,Z 540.419,A -85,B 0,C 180,E1 27051.061,E2 27051.061} C_VEL
LIN {X 0,Y 626.385,Z 518.541,A -85,B 0,C 180,E1 27048.682,E2 27048.682} C_VEL
LIN {X 0,Y 618.191,Z 499.636,A -85,B 0,C 180,E1 27046.437,E2 27046.437} C_VEL
LIN {X 0,Y 617.03,Z 496.508,A -85,B 0,C 180,E1 27046.013,E2 27046.013} C_VEL
LIN {X 0,Y 616.979,Z 496.335,A -85,B 0,C 180,E1 27042.896,E2 27042.896} C_VEL
LIN {X 0,Y 617.015,Z 496.366,A -85,B 0,C 180,E1 27039.679,E2 27039.679} C_VEL
LIN {X 0,Y 616.99,Z 496.35,A -85,B 0,C 180,E1 27036.496,E2 27036.496} C_VEL
LIN {X 0,Y 616.996,Z 496.364,A -85,B 0,C 180,E1 27033.213,E2 27033.213} C_VEL
LIN {X 0,Y 617.016,Z 496.364,A -85,B 0,C 180,E1 27030.049,E2 27030.049} C_VEL
LIN {X 0,Y 616.984,Z 496.363,A -85,B 0,C 180,E1 27026.882,E2 27026.882} C_VEL
LIN {X 0,Y 617.012,Z 496.364,A -85,B 0,C 180,E1 27023.798,E2 27023.798} C_VEL
LIN {X 0,Y 616.982,Z 496.372,A -85,B 0,C 180,E1 27020.689,E2 27020.689} C_VEL
LIN {X 0,Y 617.014,Z 496.372,A -85,B 0,C 180,E1 27017.543,E2 27017.543} C_VEL
LIN {X 0,Y 616.973,Z 496.36,A -85,B 0,C 180,E1 27014.357,E2 27014.357} C_VEL
LIN {X 0,Y 617.012,Z 496.362,A -85,B 0,C 180,E1 27011.308,E2 27011.308} C_VEL
LIN {X 0,Y 616.974,Z 496.373,A -85,B 0,C 180,E1 27008.199,E2 27008.199} C_VEL
LIN {X 0,Y 617.013,Z 496.363,A -85,B 0,C 180,E1 27005.114,E2 27005.114} C_VEL
LIN {X 0,Y 616.968,Z 496.369,A -85,B 0,C 180,E1 27001.95,E2 27001.95} C_VEL
LIN {X 0,Y 617.015,Z 496.374,A -85,B 0,C 180,E1 26998.886,E2 26998.886} C_VEL
LIN {X 0,Y 616.966,Z 496.364,A -85,B 0,C 180,E1 26995.725,E2 26995.725} C_VEL
LIN {X 0,Y 617.014,Z 496.357,A -85,B 0,C 180,E1 26992.626,E2 26992.626} C_VEL
LIN {X 0,Y 616.967,Z 496.375,A -85,B 0,C 180,E1 26989.542,E2 26989.542} C_VEL
LIN {X 0,Y 617.016,Z 496.367,A -85,B 0,C 180,E1 26986.41,E2 26986.41} C_VEL
LIN {X 0,Y 616.963,Z 496.365,A -85,B 0,C 180,E1 26983.33,E2 26983.33} C_VEL
LIN {X 0,Y 617.016,Z 496.365,A -85,B 0,C 180,E1 26980.203,E2 26980.203} C_VEL
LIN {X 0,Y 616.964,Z 496.375,A -85,B 0,C 180,E1 26977.11,E2 26977.11} C_VEL
LIN {X 0,Y 617.017,Z 496.371,A -85,B 0,C 180,E1 26974.053,E2 26974.053} C_VEL
LIN {X 0,Y 616.961,Z 496.368,A -85,B 0,C 180,E1 26971.015,E2 26971.015} C_VEL
LIN {X 0,Y 617.012,Z 496.342,A -85,B 0,C 180,E1 26968,E2 26968} C_VEL
LIN {X 0,Y 616.961,Z 496.368,A -85,B 0,C 180,E1 26964.876,E2 26964.876} C_VEL
LIN {X 0,Y 617.013,Z 496.334,A -85,B 0,C 180,E1 26961.807,E2 26961.807} C_VEL
LIN {X 0,Y 616.962,Z 496.379,A -85,B 0,C 180,E1 26958.73,E2 26958.73} C_VEL
LIN {X 0,Y 617.009,Z 496.333,A -85,B 0,C 180,E1 26955.697,E2 26955.697} C_VEL
LIN {X 0,Y 617.004,Z 496.668,A -85,B 0,C 180,E1 26954.283,E2 26954.283} C_VEL
LIN {X 0,Y 618.43,Z 500.056,A -85,B 0,C 180,E1 26953.854,E2 26953.854} C_VEL
LIN {X 0,Y 627.072,Z 519.776,A -85,B 0,C 180,E1 26951.596,E2 26951.596} C_VEL
LIN {X 0,Y 633.916,Z 536.317,A -85,B 0,C 180,E1 26949.864,E2 26949.864} C_VEL
LIN {X 0,Y 637.525,Z 542.75,A -85,B 0,C 180,E1 26949.524,E2 26949.524} C_VEL
LIN {X 0,Y 640.305,Z 557.795,A -85,B 0,C 180,E1 26949.128,E2 26949.128} C_VEL
LIN {X 0,Y 636.31,Z 799.75,A -85,B 0,C 180,E1 26945.992,E2 26945.992} C_VEL
LIN {X 0,Y 634.613,Z 921.852,A -85,B 0,C 180,E1 26944.443,E2 26944.443} C_VEL
LIN {X 0,Y 633.774,Z 946.998,A -85,B 0,C 180,E1 26943.964,E2 26943.964} C_VEL
LIN {X 0,Y 632.853,Z 969.19,A -85,B 0,C 180,E1 26943.405,E2 26943.405} C_VEL
LIN {X 0,Y 631.598,Z 994.147,A -85,B 0,C 180,E1 26942.599,E2 26942.599} C_VEL
LIN {X 0,Y 630.447,Z 1014.266,A -85,B 0,C 180,E1 26941.811,E2 26941.811} C_VEL
LIN {X 0,Y 628.9,Z 1038.244,A -85,B 0,C 180,E1 26940.687,E2 26940.687} C_VEL
LIN {X 0,Y 627.514,Z 1057.52,A -85,B 0,C 180,E1 26939.628,E2 26939.628} C_VEL
LIN {X 0,Y 625.837,Z 1079.623,A -85,B 0,C 180,E1 26938.223,E2 26938.223} C_VEL
LIN {X 0,Y 624.452,Z 1097.06,A -85,B 0,C 180,E1 26936.945,E2 26936.945} C_VEL
LIN {X 0,Y 623.11,Z 1113.621,A -85,B 0,C 180,E1 26935.572,E2 26935.572} C_VEL
LIN {X 0,Y 621.49,Z 1131.531,A -85,B 0,C 180,E1 26933.817,E2 26933.817} C_VEL
LIN {X 0,Y 620.23,Z 1146.474,A -85,B 0,C 180,E1 26932.162,E2 26932.162} C_VEL
LIN {X 0,Y 618.964,Z 1162.518,A -85,B 0,C 180,E1 26930.125,E2 26930.125} C_VEL
LIN {X 0,Y 618.033,Z 1175.408,A -85,B 0,C 180,E1 26928.252,E2 26928.252} C_VEL
LIN {X 0,Y 617.233,Z 1188.284,A -85,B 0,C 180,E1 26926.081,E2 26926.081} C_VEL
LIN {X 0,Y 616.731,Z 1198.019,A -85,B 0,C 180,E1 26924.17,E2 26924.17} C_VEL
LIN {X 0,Y 616.335,Z 1207.838,A -85,B 0,C 180,E1 26921.89,E2 26921.89} C_VEL
LIN {X 0,Y 616.097,Z 1214.859,A -85,B 0,C 180,E1 26919.893,E2 26919.893} C_VEL
LIN {X 0,Y 615.966,Z 1221.016,A -85,B 0,C 180,E1 26917.743,E2 26917.743} C_VEL
LIN {X 0,Y 615.917,Z 1225.495,A -85,B 0,C 180,E1 26915.59,E2 26915.59} C_VEL
LIN {X 0,Y 615.912,Z 1228.35,A -85,B 0,C 180,E1 26913.63,E2 26913.63} C_VEL
LIN {X 0,Y 615.908,Z 1230.214,A -85,B 0,C 180,E1 26911.209,E2 26911.209} C_VEL
LIN {X 0,Y 615.887,Z 1230.327,A -85,B 0,C 180,E1 26909.256,E2 26909.256} C_VEL
LIN {X 0,Y 615.888,Z 1229.291,A -85,B 0,C 180,E1 26907.302,E2 26907.302} C_VEL
LIN {X 0,Y 615.901,Z 1226.452,A -85,B 0,C 180,E1 26904.971,E2 26904.971} C_VEL
LIN {X 0,Y 615.968,Z 1222.689,A -85,B 0,C 180,E1 26903.007,E2 26903.007} C_VEL
LIN {X 0,Y 616.068,Z 1216.935,A -85,B 0,C 180,E1 26900.754,E2 26900.754} C_VEL
LIN {X 0,Y 616.25,Z 1209.603,A -85,B 0,C 180,E1 26898.583,E2 26898.583} C_VEL
LIN {X 0,Y 616.573,Z 1201.535,A -85,B 0,C 180,E1 26896.591,E2 26896.591} C_VEL
LIN {X 0,Y 617.092,Z 1190.862,A -85,B 0,C 180,E1 26894.397,E2 26894.397} C_VEL
LIN {X 0,Y 617.743,Z 1179.971,A -85,B 0,C 180,E1 26892.479,E2 26892.479} C_VEL
LIN {X 0,Y 618.75,Z 1165.321,A -85,B 0,C 180,E1 26890.261,E2 26890.261} C_VEL
LIN {X 0,Y 619.76,Z 1152.079,A -85,B 0,C 180,E1 26888.517,E2 26888.517} C_VEL
LIN {X 0,Y 621.254,Z 1134.309,A -85,B 0,C 180,E1 26886.476,E2 26886.476} C_VEL
LIN {X 0,Y 622.615,Z 1118.804,A -85,B 0,C 180,E1 26884.915,E2 26884.915} C_VEL
LIN {X 0,Y 624.066,Z 1102.148,A -85,B 0,C 180,E1 26883.448,E2 26883.448} C_VEL
LIN {X 0,Y 625.575,Z 1082.982,A -85,B 0,C 180,E1 26882.014,E2 26882.014} C_VEL
LIN {X 0,Y 627.118,Z 1063.014,A -85,B 0,C 180,E1 26880.694,E2 26880.694} C_VEL
LIN {X 0,Y 628.617,Z 1042.033,A -85,B 0,C 180,E1 26879.51,E2 26879.51} C_VEL
LIN {X 0,Y 630.003,Z 1021.896,A -85,B 0,C 180,E1 26878.524,E2 26878.524} C_VEL
LIN {X 0,Y 631.351,Z 999.034,A -85,B 0,C 180,E1 26877.579,E2 26877.579} C_VEL
LIN {X 0,Y 632.406,Z 978.398,A -85,B 0,C 180,E1 26876.873,E2 26876.873} C_VEL
LIN {X 0,Y 633.488,Z 953.794,A -85,B 0,C 180,E1 26876.189,E2 26876.189} C_VEL
LIN {X 0,Y 634.304,Z 931.292,A -85,B 0,C 180,E1 26875.72,E2 26875.72} C_VEL
LIN {X 0,Y 634.928,Z 906.184,A -85,B 0,C 180,E1 26875.338,E2 26875.338} C_VEL
LIN {X 0,Y 637.652,Z 712.48,A -85,B 0,C 180,E1 26872.892,E2 26872.892} C_VEL
LIN {X 0,Y 640.182,Z 556.123,A -85,B 0,C 180,E1 26870.84,E2 26870.84} C_VEL
LIN {X 0,Y 637.148,Z 541.783,A -85,B 0,C 180,E1 26870.438,E2 26870.438} C_VEL
LIN {X 0,Y 633.593,Z 535.607,A -85,B 0,C 180,E1 26870.083,E2 26870.083} C_VEL
LIN {X 0,Y 625.209,Z 515.211,A -85,B 0,C 180,E1 26867.908,E2 26867.908} C_VEL
LIN {X 0,Y 617.982,Z 499.362,A -85,B 0,C 180,E1 26866.055,E2 26866.055} C_VEL
LIN {X 0,Y 616.989,Z 496.576,A -85,B 0,C 180,E1 26865.697,E2 26865.697} C_VEL
LIN {X 0,Y 616.984,Z 496.345,A -85,B 0,C 180,E1 26862.895,E2 26862.895} C_VEL
LIN {X 0,Y 616.966,Z 496.336,A -85,B 0,C 180,E1 26859.665,E2 26859.665} C_VEL
LIN {X 0,Y 616.995,Z 496.372,A -85,B 0,C 180,E1 26856.663,E2 26856.663} C_VEL
LIN {X 0,Y 616.965,Z 496.331,A -85,B 0,C 180,E1 26853.425,E2 26853.425} C_VEL
LIN {X 0,Y 617.012,Z 496.37,A -85,B 0,C 180,E1 26850.372,E2 26850.372} C_VEL
LIN {X 0,Y 616.97,Z 496.378,A -85,B 0,C 180,E1 26847.164,E2 26847.164} C_VEL
LIN {X 0,Y 617.014,Z 496.361,A -85,B 0,C 180,E1 26844.103,E2 26844.103} C_VEL
LIN {X 0,Y 616.969,Z 496.365,A -85,B 0,C 180,E1 26840.988,E2 26840.988} C_VEL
LIN {X 0,Y 617.012,Z 496.37,A -85,B 0,C 180,E1 26837.933,E2 26837.933} C_VEL
LIN {X 0,Y 616.97,Z 496.376,A -85,B 0,C 180,E1 26834.741,E2 26834.741} C_VEL
LIN {X 0,Y 617.013,Z 496.359,A -85,B 0,C 180,E1 26831.687,E2 26831.687} C_VEL
LIN {X 0,Y 616.969,Z 496.359,A -85,B 0,C 180,E1 26828.575,E2 26828.575} C_VEL
LIN {X 0,Y 617.015,Z 496.37,A -85,B 0,C 180,E1 26825.487,E2 26825.487} C_VEL
LIN {X 0,Y 616.972,Z 496.373,A -85,B 0,C 180,E1 26822.322,E2 26822.322} C_VEL
LIN {X 0,Y 617.012,Z 496.361,A -85,B 0,C 180,E1 26819.257,E2 26819.257} C_VEL
LIN {X 0,Y 616.973,Z 496.373,A -85,B 0,C 180,E1 26816.097,E2 26816.097} C_VEL
LIN {X 0,Y 617.011,Z 496.362,A -85,B 0,C 180,E1 26813.019,E2 26813.019} C_VEL
LIN {X 0,Y 616.974,Z 496.359,A -85,B 0,C 180,E1 26809.92,E2 26809.92} C_VEL
LIN {X 0,Y 617.011,Z 496.374,A -85,B 0,C 180,E1 26806.791,E2 26806.791} C_VEL
LIN {X 0,Y 616.978,Z 496.375,A -85,B 0,C 180,E1 26803.718,E2 26803.718} C_VEL
LIN {X 0,Y 617.011,Z 496.359,A -85,B 0,C 180,E1 26800.582,E2 26800.582} C_VEL
LIN {X 0,Y 616.978,Z 496.362,A -85,B 0,C 180,E1 26797.477,E2 26797.477} C_VEL
LIN {X 0,Y 617.009,Z 496.374,A -85,B 0,C 180,E1 26794.362,E2 26794.362} C_VEL
LIN {X 0,Y 616.982,Z 496.374,A -85,B 0,C 180,E1 26791.228,E2 26791.228} C_VEL
LIN {X 0,Y 617.009,Z 496.375,A -85,B 0,C 180,E1 26788.109,E2 26788.109} C_VEL
LIN {X 0,Y 616.987,Z 496.375,A -85,B 0,C 180,E1 26784.992,E2 26784.992} C_VEL
LIN {X 0,Y 617.005,Z 496.33,A -85,B 0,C 180,E1 26781.808,E2 26781.808} C_VEL
LIN {X 0,Y 616.987,Z 496.367,A -85,B 0,C 180,E1 26778.731,E2 26778.731} C_VEL
LIN {X 0,Y 617.01,Z 496.359,A -85,B 0,C 180,E1 26775.481,E2 26775.481} C_VEL
LIN {X 0,Y 617.043,Z 496.621,A -85,B 0,C 180,E1 26773.854,E2 26773.854} C_VEL
LIN {X 0,Y 625.362,Z 516.26,A -85,B 0,C 180,E1 26771.489,E2 26771.489} C_VEL
LIN {X 0,Y 633.128,Z 535.44,A -85,B 0,C 180,E1 26769.37,E2 26769.37} C_VEL
LIN {X 0,Y 635.019,Z 540.989,A -85,B 0,C 180,E1 26768.804,E2 26768.804} C_VEL
LIN {X 0,Y 634.976,Z 541.631,A -85,B 0,C 180,E1 26768.759,E2 26768.759} C_VEL
LIN {X 0,Y 633.719,Z 547.957,A -85,B 0,C 180,E1 26768.368,E2 26768.368} C_VEL
LIN {X 0,Y 627.282,Z 565.711,A -85,B 0,C 180,E1 26767.48,E2 26767.48} C_VEL
LIN {X 0,Y 626.304,Z 571.138,A -85,B 0,C 180,E1 26767.137,E2 26767.137} C_VEL
LIN {X 0,Y 623.472,Z 615.415,A -85,B 0,C 180,E1 26764.034,E2 26764.034} C_VEL
LIN {X 0,Y 622.011,Z 642.706,A -85,B 0,C 180,E1 26762.182,E2 26762.182} C_VEL
LIN {X 0,Y 628.033,Z 676.898,A -85,B 0,C 180,E1 26761.349,E2 26761.349} C_VEL
LIN {X 0,Y 625.245,Z 950.698,A -85,B 0,C 180,E1 26758.138,E2 26758.138} C_VEL
LIN {X 0,Y 624.578,Z 972.544,A -85,B 0,C 180,E1 26757.765,E2 26757.765} C_VEL
LIN {X 0,Y 623.642,Z 992.678,A -85,B 0,C 180,E1 26757.263,E2 26757.263} C_VEL
LIN {X 0,Y 622.371,Z 1013.569,A -85,B 0,C 180,E1 26756.578,E2 26756.578} C_VEL
LIN {X 0,Y 620.994,Z 1033.25,A -85,B 0,C 180,E1 26755.768,E2 26755.768} C_VEL
LIN {X 0,Y 619.4,Z 1051.964,A -85,B 0,C 180,E1 26754.816,E2 26754.816} C_VEL
LIN {X 0,Y 617.66,Z 1070.838,A -85,B 0,C 180,E1 26753.669,E2 26753.669} C_VEL
LIN {X 0,Y 615.969,Z 1088.146,A -85,B 0,C 180,E1 26752.424,E2 26752.424} C_VEL
LIN {X 0,Y 614.251,Z 1105.185,A -85,B 0,C 180,E1 26750.984,E2 26750.984} C_VEL
LIN {X 0,Y 612.635,Z 1121.746,A -85,B 0,C 180,E1 26749.348,E2 26749.348} C_VEL
LIN {X 0,Y 611.278,Z 1136.808,A -85,B 0,C 180,E1 26747.614,E2 26747.614} C_VEL
LIN {X 0,Y 610.157,Z 1150.303,A -85,B 0,C 180,E1 26745.785,E2 26745.785} C_VEL
LIN {X 0,Y 609.29,Z 1162.363,A -85,B 0,C 180,E1 26743.862,E2 26743.862} C_VEL
LIN {X 0,Y 608.676,Z 1172.976,A -85,B 0,C 180,E1 26741.849,E2 26741.849} C_VEL
LIN {X 0,Y 608.297,Z 1181.727,A -85,B 0,C 180,E1 26739.843,E2 26739.843} C_VEL
LIN {X 0,Y 608.063,Z 1188.617,A -85,B 0,C 180,E1 26737.844,E2 26737.844} C_VEL
LIN {X 0,Y 607.952,Z 1194.336,A -85,B 0,C 180,E1 26735.663,E2 26735.663} C_VEL
LIN {X 0,Y 607.921,Z 1197.976,A -85,B 0,C 180,E1 26733.678,E2 26733.678} C_VEL
LIN {X 0,Y 607.911,Z 1199.97,A -85,B 0,C 180,E1 26731.697,E2 26731.697} C_VEL
LIN {X 0,Y 607.902,Z 1200.515,A -85,B 0,C 180,E1 26729.529,E2 26729.529} C_VEL
LIN {X 0,Y 607.914,Z 1199.425,A -85,B 0,C 180,E1 26727.455,E2 26727.455} C_VEL
LIN {X 0,Y 607.933,Z 1196.719,A -85,B 0,C 180,E1 26725.472,E2 26725.472} C_VEL
LIN {X 0,Y 607.986,Z 1192.066,A -85,B 0,C 180,E1 26723.295,E2 26723.295} C_VEL
LIN {X 0,Y 608.148,Z 1186.215,A -85,B 0,C 180,E1 26721.3,E2 26721.3} C_VEL
LIN {X 0,Y 608.417,Z 1178.544,A -85,B 0,C 180,E1 26719.298,E2 26719.298} C_VEL
LIN {X 0,Y 608.882,Z 1169.073,A -85,B 0,C 180,E1 26717.28,E2 26717.28} C_VEL
LIN {X 0,Y 609.571,Z 1158.37,A -85,B 0,C 180,E1 26715.369,E2 26715.369} C_VEL
LIN {X 0,Y 610.471,Z 1146.201,A -85,B 0,C 180,E1 26713.54,E2 26713.54} C_VEL
LIN {X 0,Y 611.634,Z 1132.428,A -85,B 0,C 180,E1 26711.771,E2 26711.771} C_VEL
LIN {X 0,Y 613.042,Z 1117.609,A -85,B 0,C 180,E1 26710.125,E2 26710.125} C_VEL
LIN {X 0,Y 614.592,Z 1101.9,A -85,B 0,C 180,E1 26708.628,E2 26708.628} C_VEL
LIN {X 0,Y 616.278,Z 1084.84,A -85,B 0,C 180,E1 26707.235,E2 26707.235} C_VEL
LIN {X 0,Y 618.04,Z 1067.065,A -85,B 0,C 180,E1 26705.991,E2 26705.991} C_VEL
LIN {X 0,Y 619.654,Z 1049.161,A -85,B 0,C 180,E1 26704.94,E2 26704.94} C_VEL
LIN {X 0,Y 621.312,Z 1028.6,A -85,B 0,C 180,E1 26703.939,E2 26703.939} C_VEL
LIN {X 0,Y 622.742,Z 1008.818,A -85,B 0,C 180,E1 26703.156,E2 26703.156} C_VEL
LIN {X 0,Y 623.866,Z 988.06,A -85,B 0,C 180,E1 26702.518,E2 26702.518} C_VEL
LIN {X 0,Y 624.826,Z 965.471,A -85,B 0,C 180,E1 26702.007,E2 26702.007} C_VEL
LIN {X 0,Y 625.406,Z 943.238,A -85,B 0,C 180,E1 26701.673,E2 26701.673} C_VEL
LIN {X 0,Y 628.014,Z 675.579,A -85,B 0,C 180,E1 26698.54,E2 26698.54} C_VEL
LIN {X 0,Y 621.958,Z 641.828,A -85,B 0,C 180,E1 26697.688,E2 26697.688} C_VEL
LIN {X 0,Y 624.834,Z 593.891,A -85,B 0,C 180,E1 26694.376,E2 26694.376} C_VEL
LIN {X 0,Y 627.849,Z 549.094,A -85,B 0,C 180,E1 26691.196,E2 26691.196} C_VEL
LIN {X 0,Y 628.149,Z 543.779,A -85,B 0,C 180,E1 26690.808,E2 26690.808} C_VEL
LIN {X 0,Y 619.772,Z 522.561,A -85,B 0,C 180,E1 26688.467,E2 26688.467} C_VEL
LIN {X 0,Y 611.927,Z 504.361,A -85,B 0,C 180,E1 26686.278,E2 26686.278} C_VEL
LIN {X 0,Y 609.081,Z 497.585,A -85,B 0,C 180,E1 26685.399,E2 26685.399} C_VEL
LIN {X 0,Y 609.066,Z 497.321,A -85,B 0,C 180,E1 26682.377,E2 26682.377} C_VEL
LIN {X 0,Y 609.044,Z 497.34,A -85,B 0,C 180,E1 26679.203,E2 26679.203} C_VEL
LIN {X 0,Y 609.071,Z 497.344,A -85,B 0,C 180,E1 26676.112,E2 26676.112} C_VEL
LIN {X 0,Y 609.041,Z 497.355,A -85,B 0,C 180,E1 26672.917,E2 26672.917} C_VEL
LIN {X 0,Y 609.075,Z 497.353,A -85,B 0,C 180,E1 26669.83,E2 26669.83} C_VEL
LIN {X 0,Y 609.039,Z 497.351,A -85,B 0,C 180,E1 26666.734,E2 26666.734} C_VEL
LIN {X 0,Y 609.073,Z 497.349,A -85,B 0,C 180,E1 26663.614,E2 26663.614} C_VEL
LIN {X 0,Y 609.037,Z 497.363,A -85,B 0,C 180,E1 26660.469,E2 26660.469} C_VEL
LIN {X 0,Y 609.076,Z 497.363,A -85,B 0,C 180,E1 26657.384,E2 26657.384} C_VEL
LIN {X 0,Y 609.033,Z 497.349,A -85,B 0,C 180,E1 26654.257,E2 26654.257} C_VEL
LIN {X 0,Y 609.073,Z 497.348,A -85,B 0,C 180,E1 26651.17,E2 26651.17} C_VEL
LIN {X 0,Y 609.033,Z 497.364,A -85,B 0,C 180,E1 26648.022,E2 26648.022} C_VEL
LIN {X 0,Y 609.073,Z 497.355,A -85,B 0,C 180,E1 26644.897,E2 26644.897} C_VEL
LIN {X 0,Y 609.029,Z 497.358,A -85,B 0,C 180,E1 26641.788,E2 26641.788} C_VEL
LIN {X 0,Y 609.076,Z 497.36,A -85,B 0,C 180,E1 26638.668,E2 26638.668} C_VEL
LIN {X 0,Y 609.029,Z 497.353,A -85,B 0,C 180,E1 26635.574,E2 26635.574} C_VEL
LIN {X 0,Y 609.078,Z 497.343,A -85,B 0,C 180,E1 26632.453,E2 26632.453} C_VEL
LIN {X 0,Y 609.032,Z 497.366,A -85,B 0,C 180,E1 26629.309,E2 26629.309} C_VEL
LIN {X 0,Y 609.076,Z 497.359,A -85,B 0,C 180,E1 26626.132,E2 26626.132} C_VEL
LIN {X 0,Y 609.029,Z 497.352,A -85,B 0,C 180,E1 26623.106,E2 26623.106} C_VEL
LIN {X 0,Y 609.065,Z 497.351,A -85,B 0,C 180,E1 26619.886,E2 26619.886} C_VEL
LIN {X 0,Y 609.036,Z 497.366,A -85,B 0,C 180,E1 26616.795,E2 26616.795} C_VEL
LIN {X 0,Y 609.045,Z 497.362,A -85,B 0,C 180,E1 26613.472,E2 26613.472} C_VEL
LIN {X 0,Y 609.046,Z 497.36,A -85,B 0,C 180,E1 26610.469,E2 26610.469} C_VEL
LIN {X 0,Y 609.03,Z 497.32,A -85,B 0,C 180,E1 26607.195,E2 26607.195} C_VEL
LIN {X 0,Y 609.06,Z 497.363,A -85,B 0,C 180,E1 26604.12,E2 26604.12} C_VEL
LIN {X 0,Y 609.021,Z 497.319,A -85,B 0,C 180,E1 26600.916,E2 26600.916} C_VEL
LIN {X 0,Y 609.062,Z 497.353,A -85,B 0,C 180,E1 26597.904,E2 26597.904} C_VEL
LIN {X 0,Y 609.068,Z 497.565,A -85,B 0,C 180,E1 26594.954,E2 26594.954} C_VEL
LIN {X 0,Y 610.301,Z 500.817,A -85,B 0,C 180,E1 26594.523,E2 26594.523} C_VEL
LIN {X 0,Y 617.896,Z 517.62,A -85,B 0,C 180,E1 26592.515,E2 26592.515} C_VEL
LIN {X 0,Y 626.112,Z 537.244,A -85,B 0,C 180,E1 26590.38,E2 26590.38} C_VEL
LIN {X 0,Y 631.493,Z 546.695,A -85,B 0,C 180,E1 26589.866,E2 26589.866} C_VEL
LIN {X 0,Y 633.775,Z 559.419,A -85,B 0,C 180,E1 26589.529,E2 26589.529} C_VEL
LIN {X 0,Y 629.206,Z 812.746,A -85,B 0,C 180,E1 26586.193,E2 26586.193} C_VEL
LIN {X 0,Y 627.521,Z 921.821,A -85,B 0,C 180,E1 26584.783,E2 26584.783} C_VEL
LIN {X 0,Y 626.635,Z 946.911,A -85,B 0,C 180,E1 26584.298,E2 26584.298} C_VEL
LIN {X 0,Y 625.665,Z 968.893,A -85,B 0,C 180,E1 26583.737,E2 26583.737} C_VEL
LIN {X 0,Y 624.328,Z 994.021,A -85,B 0,C 180,E1 26582.918,E2 26582.918} C_VEL
LIN {X 0,Y 623.012,Z 1016.153,A -85,B 0,C 180,E1 26582.039,E2 26582.039} C_VEL
LIN {X 0,Y 621.45,Z 1039.198,A -85,B 0,C 180,E1 26580.939,E2 26580.939} C_VEL
LIN {X 0,Y 620.099,Z 1057.26,A -85,B 0,C 180,E1 26579.937,E2 26579.937} C_VEL
LIN {X 0,Y 618.353,Z 1079.022,A -85,B 0,C 180,E1 26578.543,E2 26578.543} C_VEL
LIN {X 0,Y 616.901,Z 1096.398,A -85,B 0,C 180,E1 26577.259,E2 26577.259} C_VEL
LIN {X 0,Y 615.36,Z 1114.997,A -85,B 0,C 180,E1 26575.711,E2 26575.711} C_VEL
LIN {X 0,Y 613.895,Z 1131.794,A -85,B 0,C 180,E1 26574.093,E2 26574.093} C_VEL
LIN {X 0,Y 612.727,Z 1144.782,A -85,B 0,C 180,E1 26572.65,E2 26572.65} C_VEL
LIN {X 0,Y 611.398,Z 1160.415,A -85,B 0,C 180,E1 26570.685,E2 26570.685} C_VEL
LIN {X 0,Y 610.336,Z 1173.879,A -85,B 0,C 180,E1 26568.729,E2 26568.729} C_VEL
LIN {X 0,Y 609.462,Z 1186.738,A -85,B 0,C 180,E1 26566.586,E2 26566.586} C_VEL
LIN {X 0,Y 608.853,Z 1197.1,A -85,B 0,C 180,E1 26564.552,E2 26564.552} C_VEL
LIN {X 0,Y 608.413,Z 1206.774,A -85,B 0,C 180,E1 26562.336,E2 26562.336} C_VEL
LIN {X 0,Y 608.134,Z 1214.211,A -85,B 0,C 180,E1 26560.228,E2 26560.228} C_VEL
LIN {X 0,Y 608.031,Z 1219.746,A -85,B 0,C 180,E1 26558.32,E2 26558.32} C_VEL
LIN {X 0,Y 607.942,Z 1225.016,A -85,B 0,C 180,E1 26555.947,E2 26555.947} C_VEL
LIN {X 0,Y 607.915,Z 1228.123,A -85,B 0,C 180,E1 26553.867,E2 26553.867} C_VEL
LIN {X 0,Y 607.897,Z 1230.103,A -85,B 0,C 180,E1 26551.602,E2 26551.602} C_VEL
LIN {X 0,Y 607.884,Z 1230.372,A -85,B 0,C 180,E1 26549.435,E2 26549.435} C_VEL
LIN {X 0,Y 607.895,Z 1229.427,A -85,B 0,C 180,E1 26547.455,E2 26547.455} C_VEL
LIN {X 0,Y 607.912,Z 1226.928,A -85,B 0,C 180,E1 26545.188,E2 26545.188} C_VEL
LIN {X 0,Y 607.965,Z 1223.102,A -85,B 0,C 180,E1 26543.105,E2 26543.105} C_VEL
LIN {X 0,Y 608.04,Z 1218.22,A -85,B 0,C 180,E1 26541.108,E2 26541.108} C_VEL
LIN {X 0,Y 608.248,Z 1210.661,A -85,B 0,C 180,E1 26538.719,E2 26538.719} C_VEL
LIN {X 0,Y 608.58,Z 1202.75,A -85,B 0,C 180,E1 26536.702,E2 26536.702} C_VEL
LIN {X 0,Y 609.121,Z 1192.405,A -85,B 0,C 180,E1 26534.481,E2 26534.481} C_VEL
LIN {X 0,Y 609.822,Z 1181.116,A -85,B 0,C 180,E1 26532.441,E2 26532.441} C_VEL
LIN {X 0,Y 610.778,Z 1168.121,A -85,B 0,C 180,E1 26530.392,E2 26530.392} C_VEL
LIN {X 0,Y 611.884,Z 1154.388,A -85,B 0,C 180,E1 26528.529,E2 26528.529} C_VEL
LIN {X 0,Y 613.288,Z 1138.865,A -85,B 0,C 180,E1 26526.661,E2 26526.661} C_VEL
LIN {X 0,Y 614.66,Z 1122.93,A -85,B 0,C 180,E1 26525.031,E2 26525.031} C_VEL
LIN {X 0,Y 616.059,Z 1106.328,A -85,B 0,C 180,E1 26523.544,E2 26523.544} C_VEL
LIN {X 0,Y 617.873,Z 1084.975,A -85,B 0,C 180,E1 26521.88,E2 26521.88} C_VEL
LIN {X 0,Y 619.391,Z 1066.214,A -85,B 0,C 180,E1 26520.611,E2 26520.611} C_VEL
LIN {X 0,Y 621.142,Z 1043.283,A -85,B 0,C 180,E1 26519.274,E2 26519.274} C_VEL
LIN {X 0,Y 622.501,Z 1023.991,A -85,B 0,C 180,E1 26518.317,E2 26518.317} C_VEL
LIN {X 0,Y 624.024,Z 999.654,A -85,B 0,C 180,E1 26517.291,E2 26517.291} C_VEL
LIN {X 0,Y 625.186,Z 978.061,A -85,B 0,C 180,E1 26516.542,E2 26516.542} C_VEL
LIN {X 0,Y 626.357,Z 953.113,A -85,B 0,C 180,E1 26515.844,E2 26515.844} C_VEL
LIN {X 0,Y 627.22,Z 930.82,A -85,B 0,C 180,E1 26515.375,E2 26515.375} C_VEL
LIN {X 0,Y 627.88,Z 905.011,A -85,B 0,C 180,E1 26514.981,E2 26514.981} C_VEL
LIN {X 0,Y 631.273,Z 693.01,A -85,B 0,C 180,E1 26512.237,E2 26512.237} C_VEL
LIN {X 0,Y 633.657,Z 557.734,A -85,B 0,C 180,E1 26510.438,E2 26510.438} C_VEL
LIN {X 0,Y 631.077,Z 545.613,A -85,B 0,C 180,E1 26510.091,E2 26510.091} C_VEL
LIN {X 0,Y 625.86,Z 536.676,A -85,B 0,C 180,E1 26509.576,E2 26509.576} C_VEL
LIN {X 0,Y 617.326,Z 516.285,A -85,B 0,C 180,E1 26507.337,E2 26507.337} C_VEL
LIN {X 0,Y 610.21,Z 500.668,A -85,B 0,C 180,E1 26505.463,E2 26505.463} C_VEL
LIN {X 0,Y 609.066,Z 497.535,A -85,B 0,C 180,E1 26505.037,E2 26505.037} C_VEL
LIN {X 0,Y 609.048,Z 497.359,A -85,B 0,C 180,E1 26501.927,E2 26501.927} C_VEL
LIN {X 0,Y 609.034,Z 497.318,A -85,B 0,C 180,E1 26498.907,E2 26498.907} C_VEL
LIN {X 0,Y 609.041,Z 497.36,A -85,B 0,C 180,E1 26495.646,E2 26495.646} C_VEL
LIN {X 0,Y 609.049,Z 497.321,A -85,B 0,C 180,E1 26492.581,E2 26492.581} C_VEL
LIN {X 0,Y 609.034,Z 497.359,A -85,B 0,C 180,E1 26489.338,E2 26489.338} C_VEL
LIN {X 0,Y 609.065,Z 497.361,A -85,B 0,C 180,E1 26486.312,E2 26486.312} C_VEL
LIN {X 0,Y 609.032,Z 497.366,A -85,B 0,C 180,E1 26483.103,E2 26483.103} C_VEL
LIN {X 0,Y 609.069,Z 497.351,A -85,B 0,C 180,E1 26480.067,E2 26480.067} C_VEL
LIN {X 0,Y 609.03,Z 497.353,A -85,B 0,C 180,E1 26476.839,E2 26476.839} C_VEL
LIN {X 0,Y 609.078,Z 497.359,A -85,B 0,C 180,E1 26473.771,E2 26473.771} C_VEL
LIN {X 0,Y 609.032,Z 497.364,A -85,B 0,C 180,E1 26470.596,E2 26470.596} C_VEL
LIN {X 0,Y 609.074,Z 497.343,A -85,B 0,C 180,E1 26467.452,E2 26467.452} C_VEL
LIN {X 0,Y 609.032,Z 497.351,A -85,B 0,C 180,E1 26464.331,E2 26464.331} C_VEL
LIN {X 0,Y 609.074,Z 497.36,A -85,B 0,C 180,E1 26461.223,E2 26461.223} C_VEL
LIN {X 0,Y 609.034,Z 497.358,A -85,B 0,C 180,E1 26458.118,E2 26458.118} C_VEL
LIN {X 0,Y 609.072,Z 497.354,A -85,B 0,C 180,E1 26455.008,E2 26455.008} C_VEL
LIN {X 0,Y 609.037,Z 497.363,A -85,B 0,C 180,E1 26451.868,E2 26451.868} C_VEL
LIN {X 0,Y 609.072,Z 497.348,A -85,B 0,C 180,E1 26448.734,E2 26448.734} C_VEL
LIN {X 0,Y 609.039,Z 497.348,A -85,B 0,C 180,E1 26445.604,E2 26445.604} C_VEL
LIN {X 0,Y 609.075,Z 497.361,A -85,B 0,C 180,E1 26442.418,E2 26442.418} C_VEL
LIN {X 0,Y 609.051,Z 497.361,A -85,B 0,C 180,E1 26439.23,E2 26439.23} C_VEL
LIN {X 0,Y 609.066,Z 497.357,A -85,B 0,C 180,E1 26435.975,E2 26435.975} C_VEL
LIN {X 0,Y 609.071,Z 497.349,A -85,B 0,C 180,E1 26432.74,E2 26432.74} C_VEL
LIN {X 0,Y 609.049,Z 497.356,A -85,B 0,C 180,E1 26429.516,E2 26429.516} C_VEL
LIN {X 0,Y 609.07,Z 497.351,A -85,B 0,C 180,E1 26426.335,E2 26426.335} C_VEL
LIN {X 0,Y 609.042,Z 497.332,A -85,B 0,C 180,E1 26423.185,E2 26423.185} C_VEL
LIN {X 0,Y 609.069,Z 497.358,A -85,B 0,C 180,E1 26420.052,E2 26420.052} C_VEL
LIN {X 0,Y 609.044,Z 497.321,A -85,B 0,C 180,E1 26416.924,E2 26416.924} C_VEL
LIN {X 0,Y 609.089,Z 497.579,A -85,B 0,C 180,E1 26414.503,E2 26414.503} C_VEL
LIN {X 0,Y 612.324,Z 505.06,A -85,B 0,C 180,E1 26413.529,E2 26413.529} C_VEL
LIN {X 0,Y 621.533,Z 526.843,A -85,B 0,C 180,E1 26410.947,E2 26410.947} C_VEL
LIN {X 0,Y 628.186,Z 544.075,A -85,B 0,C 180,E1 26409.072,E2 26409.072} C_VEL
LIN {X 0,Y 626.304,Z 571.138,A -85,B 0,C 180,E1 26407.137,E2 26407.137} C_VEL
LIN {X 0,Y 625.062,Z 577.485,A -85,B 0,C 180,E1 26406.744,E2 26406.744} C_VEL
LIN {X 0,Y 618.552,Z 595.258,A -85,B 0,C 180,E1 26405.85,E2 26405.85} C_VEL
LIN {X 0,Y 617.533,Z 600.721,A -85,B 0,C 180,E1 26405.507,E2 26405.507} C_VEL
LIN {X 0,Y 615.042,Z 641.728,A -85,B 0,C 180,E1 26402.665,E2 26402.665} C_VEL
LIN {X 0,Y 621.457,Z 678.278,A -85,B 0,C 180,E1 26401.755,E2 26401.755} C_VEL
LIN {X 0,Y 618.475,Z 952.278,A -85,B 0,C 180,E1 26398.517,E2 26398.517} C_VEL
LIN {X 0,Y 617.674,Z 975.39,A -85,B 0,C 180,E1 26398.099,E2 26398.099} C_VEL
LIN {X 0,Y 616.685,Z 995.741,A -85,B 0,C 180,E1 26397.574,E2 26397.574} C_VEL
LIN {X 0,Y 615.28,Z 1016.612,A -85,B 0,C 180,E1 26396.857,E2 26396.857} C_VEL
LIN {X 0,Y 613.658,Z 1037.818,A -85,B 0,C 180,E1 26395.938,E2 26395.938} C_VEL
LIN {X 0,Y 611.969,Z 1056.922,A -85,B 0,C 180,E1 26394.931,E2 26394.931} C_VEL
LIN {X 0,Y 610.175,Z 1075.073,A -85,B 0,C 180,E1 26393.772,E2 26393.772} C_VEL
LIN {X 0,Y 608.229,Z 1093.693,A -85,B 0,C 180,E1 26392.368,E2 26392.368} C_VEL
LIN {X 0,Y 606.49,Z 1110.166,A -85,B 0,C 180,E1 26390.904,E2 26390.904} C_VEL
LIN {X 0,Y 604.806,Z 1125.812,A -85,B 0,C 180,E1 26389.265,E2 26389.265} C_VEL
LIN {X 0,Y 603.337,Z 1140.61,A -85,B 0,C 180,E1 26387.455,E2 26387.455} C_VEL
LIN {X 0,Y 602.197,Z 1153.561,A -85,B 0,C 180,E1 26385.603,E2 26385.603} C_VEL
LIN {X 0,Y 601.323,Z 1165.141,A -85,B 0,C 180,E1 26383.657,E2 26383.657} C_VEL
LIN {X 0,Y 600.704,Z 1174.785,A -85,B 0,C 180,E1 26381.716,E2 26381.716} C_VEL
LIN {X 0,Y 600.286,Z 1183.573,A -85,B 0,C 180,E1 26379.566,E2 26379.566} C_VEL
LIN {X 0,Y 600.069,Z 1190.299,A -85,B 0,C 180,E1 26377.498,E2 26377.498} C_VEL
LIN {X 0,Y 599.963,Z 1195.196,A -85,B 0,C 180,E1 26375.451,E2 26375.451} C_VEL
LIN {X 0,Y 599.919,Z 1198.761,A -85,B 0,C 180,E1 26373.248,E2 26373.248} C_VEL
LIN {X 0,Y 599.907,Z 1200.512,A -85,B 0,C 180,E1 26371.242,E2 26371.242} C_VEL
LIN {X 0,Y 599.91,Z 1200.655,A -85,B 0,C 180,E1 26369.236,E2 26369.236} C_VEL
LIN {X 0,Y 599.919,Z 1199.198,A -85,B 0,C 180,E1 26367.038,E2 26367.038} C_VEL
LIN {X 0,Y 599.94,Z 1196.333,A -85,B 0,C 180,E1 26365.028,E2 26365.028} C_VEL
LIN {X 0,Y 600.015,Z 1191.851,A -85,B 0,C 180,E1 26363.013,E2 26363.013} C_VEL
LIN {X 0,Y 600.215,Z 1185.528,A -85,B 0,C 180,E1 26360.894,E2 26360.894} C_VEL
LIN {X 0,Y 600.557,Z 1177.775,A -85,B 0,C 180,E1 26358.865,E2 26358.865} C_VEL
LIN {X 0,Y 601.072,Z 1168.631,A -85,B 0,C 180,E1 26356.925,E2 26356.925} C_VEL
LIN {X 0,Y 601.856,Z 1157.769,A -85,B 0,C 180,E1 26354.98,E2 26354.98} C_VEL
LIN {X 0,Y 602.961,Z 1144.927,A -85,B 0,C 180,E1 26353.031,E2 26353.031} C_VEL
LIN {X 0,Y 604.254,Z 1131.224,A -85,B 0,C 180,E1 26351.276,E2 26351.276} C_VEL
LIN {X 0,Y 605.797,Z 1116.261,A -85,B 0,C 180,E1 26349.62,E2 26349.62} C_VEL
LIN {X 0,Y 607.535,Z 1100.495,A -85,B 0,C 180,E1 26348.114,E2 26348.114} C_VEL
LIN {X 0,Y 609.277,Z 1083.737,A -85,B 0,C 180,E1 26346.76,E2 26346.76} C_VEL
LIN {X 0,Y 611.146,Z 1065.396,A -85,B 0,C 180,E1 26345.497,E2 26345.497} C_VEL
LIN {X 0,Y 612.851,Z 1047.175,A -85,B 0,C 180,E1 26344.441,E2 26344.441} C_VEL
LIN {X 0,Y 614.472,Z 1027.663,A -85,B 0,C 180,E1 26343.506,E2 26343.506} C_VEL
LIN {X 0,Y 615.974,Z 1007.17,A -85,B 0,C 180,E1 26342.706,E2 26342.706} C_VEL
LIN {X 0,Y 617.139,Z 986.637,A -85,B 0,C 180,E1 26342.081,E2 26342.081} C_VEL
LIN {X 0,Y 618.098,Z 964.828,A -85,B 0,C 180,E1 26341.596,E2 26341.596} C_VEL
LIN {X 0,Y 618.689,Z 942.337,A -85,B 0,C 180,E1 26341.262,E2 26341.262} C_VEL
LIN {X 0,Y 621.443,Z 676.97,A -85,B 0,C 180,E1 26338.133,E2 26338.133} C_VEL
LIN {X 0,Y 614.995,Z 640.794,A -85,B 0,C 180,E1 26337.2,E2 26337.2} C_VEL
LIN {X 0,Y 618.022,Z 593.937,A -85,B 0,C 180,E1 26333.922,E2 26333.922} C_VEL
LIN {X 0,Y 621.295,Z 548.374,A -85,B 0,C 180,E1 26330.649,E2 26330.649} C_VEL
LIN {X 0,Y 620.994,Z 546.358,A -85,B 0,C 180,E1 26330.468,E2 26330.468} C_VEL
LIN {X 0,Y 613.169,Z 526.601,A -85,B 0,C 180,E1 26328.249,E2 26328.249} C_VEL
LIN {X 0,Y 605.614,Z 508.958,A -85,B 0,C 180,E1 26326.099,E2 26326.099} C_VEL
LIN {X 0,Y 601.159,Z 498.651,A -85,B 0,C 180,E1 26324.749,E2 26324.749} C_VEL
LIN {X 0,Y 601.106,Z 498.31,A -85,B 0,C 180,E1 26323.374,E2 26323.374} C_VEL
LIN {X 0,Y 601.137,Z 498.351,A -85,B 0,C 180,E1 26320.194,E2 26320.194} C_VEL
LIN {X 0,Y 601.099,Z 498.313,A -85,B 0,C 180,E1 26317.02,E2 26317.02} C_VEL
LIN {X 0,Y 601.134,Z 498.341,A -85,B 0,C 180,E1 26313.864,E2 26313.864} C_VEL
LIN {X 0,Y 601.1,Z 498.348,A -85,B 0,C 180,E1 26310.687,E2 26310.687} C_VEL
LIN {X 0,Y 601.135,Z 498.341,A -85,B 0,C 180,E1 26307.543,E2 26307.543} C_VEL
LIN {X 0,Y 601.102,Z 498.355,A -85,B 0,C 180,E1 26304.364,E2 26304.364} C_VEL
LIN {X 0,Y 601.137,Z 498.348,A -85,B 0,C 180,E1 26301.158,E2 26301.158} C_VEL
LIN {X 0,Y 601.113,Z 498.343,A -85,B 0,C 180,E1 26297.931,E2 26297.931} C_VEL
LIN {X 0,Y 601.11,Z 498.334,A -85,B 0,C 180,E1 26294.646,E2 26294.646} C_VEL
LIN {X 0,Y 601.127,Z 498.344,A -85,B 0,C 180,E1 26291.514,E2 26291.514} C_VEL
LIN {X 0,Y 601.098,Z 498.351,A -85,B 0,C 180,E1 26288.226,E2 26288.226} C_VEL
LIN {X 0,Y 601.135,Z 498.338,A -85,B 0,C 180,E1 26285.153,E2 26285.153} C_VEL
LIN {X 0,Y 601.092,Z 498.346,A -85,B 0,C 180,E1 26282.002,E2 26282.002} C_VEL
LIN {X 0,Y 601.138,Z 498.352,A -85,B 0,C 180,E1 26278.856,E2 26278.856} C_VEL
LIN {X 0,Y 601.089,Z 498.341,A -85,B 0,C 180,E1 26275.707,E2 26275.707} C_VEL
LIN {X 0,Y 601.138,Z 498.332,A -85,B 0,C 180,E1 26272.545,E2 26272.545} C_VEL
LIN {X 0,Y 601.091,Z 498.354,A -85,B 0,C 180,E1 26269.442,E2 26269.442} C_VEL
LIN {X 0,Y 601.139,Z 498.347,A -85,B 0,C 180,E1 26266.24,E2 26266.24} C_VEL
LIN {X 0,Y 601.089,Z 498.34,A -85,B 0,C 180,E1 26263.175,E2 26263.175} C_VEL
LIN {X 0,Y 601.131,Z 498.339,A -85,B 0,C 180,E1 26259.962,E2 26259.962} C_VEL
LIN {X 0,Y 601.092,Z 498.355,A -85,B 0,C 180,E1 26256.885,E2 26256.885} C_VEL
LIN {X 0,Y 601.119,Z 498.351,A -85,B 0,C 180,E1 26253.633,E2 26253.633} C_VEL
LIN {X 0,Y 601.095,Z 498.348,A -85,B 0,C 180,E1 26250.612,E2 26250.612} C_VEL
LIN {X 0,Y 601.097,Z 498.306,A -85,B 0,C 180,E1 26247.274,E2 26247.274} C_VEL
LIN {X 0,Y 601.118,Z 498.351,A -85,B 0,C 180,E1 26244.161,E2 26244.161} C_VEL
LIN {X 0,Y 601.082,Z 498.306,A -85,B 0,C 180,E1 26240.916,E2 26240.916} C_VEL
LIN {X 0,Y 601.124,Z 498.339,A -85,B 0,C 180,E1 26237.888,E2 26237.888} C_VEL
LIN {X 0,Y 601.17,Z 498.571,A -85,B 0,C 180,E1 26235.608,E2 26235.608} C_VEL
LIN {X 0,Y 602.77,Z 502.345,A -85,B 0,C 180,E1 26235.096,E2 26235.096} C_VEL
LIN {X 0,Y 611.43,Z 521.754,A -85,B 0,C 180,E1 26232.737,E2 26232.737} C_VEL
LIN {X 0,Y 618.434,Z 538.364,A -85,B 0,C 180,E1 26230.899,E2 26230.899} C_VEL
LIN {X 0,Y 625.487,Z 550.646,A -85,B 0,C 180,E1 26230.215,E2 26230.215} C_VEL
LIN {X 0,Y 627.281,Z 561.099,A -85,B 0,C 180,E1 26229.938,E2 26229.938} C_VEL
LIN {X 0,Y 622.333,Z 815.768,A -85,B 0,C 180,E1 26226.539,E2 26226.539} C_VEL
LIN {X 0,Y 620.447,Z 922.294,A -85,B 0,C 180,E1 26225.123,E2 26225.123} C_VEL
LIN {X 0,Y 619.505,Z 946.996,A -85,B 0,C 180,E1 26224.634,E2 26224.634} C_VEL
LIN {X 0,Y 618.503,Z 968.482,A -85,B 0,C 180,E1 26224.08,E2 26224.08} C_VEL
LIN {X 0,Y 617.141,Z 992.982,A -85,B 0,C 180,E1 26223.277,E2 26223.277} C_VEL
LIN {X 0,Y 615.743,Z 1014.911,A -85,B 0,C 180,E1 26222.402,E2 26222.402} C_VEL
LIN {X 0,Y 614.119,Z 1038.171,A -85,B 0,C 180,E1 26221.29,E2 26221.29} C_VEL
LIN {X 0,Y 612.647,Z 1057.204,A -85,B 0,C 180,E1 26220.23,E2 26220.23} C_VEL
LIN {X 0,Y 610.831,Z 1079.127,A -85,B 0,C 180,E1 26218.82,E2 26218.82} C_VEL
LIN {X 0,Y 609.245,Z 1097.252,A -85,B 0,C 180,E1 26217.462,E2 26217.462} C_VEL
LIN {X 0,Y 607.536,Z 1116.63,A -85,B 0,C 180,E1 26215.807,E2 26215.807} C_VEL
LIN {X 0,Y 606.102,Z 1132.484,A -85,B 0,C 180,E1 26214.253,E2 26214.253} C_VEL
LIN {X 0,Y 604.709,Z 1148.786,A -85,B 0,C 180,E1 26212.454,E2 26212.454} C_VEL
LIN {X 0,Y 603.488,Z 1162.514,A -85,B 0,C 180,E1 26210.665,E2 26210.665} C_VEL
LIN {X 0,Y 602.442,Z 1175.147,A -85,B 0,C 180,E1 26208.782,E2 26208.782} C_VEL
LIN {X 0,Y 601.483,Z 1188.281,A -85,B 0,C 180,E1 26206.514,E2 26206.514} C_VEL
LIN {X 0,Y 600.888,Z 1198.017,A -85,B 0,C 180,E1 26204.552,E2 26204.552} C_VEL
LIN {X 0,Y 600.405,Z 1208.025,A -85,B 0,C 180,E1 26202.158,E2 26202.158} C_VEL
LIN {X 0,Y 600.137,Z 1214.817,A -85,B 0,C 180,E1 26200.172,E2 26200.172} C_VEL
LIN {X 0,Y 599.99,Z 1221.017,A -85,B 0,C 180,E1 26197.95,E2 26197.95} C_VEL
LIN {X 0,Y 599.929,Z 1225.519,A -85,B 0,C 180,E1 26195.724,E2 26195.724} C_VEL
LIN {X 0,Y 599.913,Z 1228.35,A -85,B 0,C 180,E1 26193.727,E2 26193.727} C_VEL
LIN {X 0,Y 599.903,Z 1230.19,A -85,B 0,C 180,E1 26191.337,E2 26191.337} C_VEL
LIN {X 0,Y 599.884,Z 1230.349,A -85,B 0,C 180,E1 26189.331,E2 26189.331} C_VEL
LIN {X 0,Y 599.89,Z 1229.359,A -85,B 0,C 180,E1 26187.325,E2 26187.325} C_VEL
LIN {X 0,Y 599.903,Z 1226.611,A -85,B 0,C 180,E1 26184.932,E2 26184.932} C_VEL
LIN {X 0,Y 599.97,Z 1222.896,A -85,B 0,C 180,E1 26182.916,E2 26182.916} C_VEL
LIN {X 0,Y 600.074,Z 1217.712,A -85,B 0,C 180,E1 26180.796,E2 26180.796} C_VEL
LIN {X 0,Y 600.296,Z 1210.308,A -85,B 0,C 180,E1 26178.471,E2 26178.471} C_VEL
LIN {X 0,Y 600.649,Z 1202.461,A -85,B 0,C 180,E1 26176.454,E2 26176.454} C_VEL
LIN {X 0,Y 601.278,Z 1191.374,A -85,B 0,C 180,E1 26174.075,E2 26174.075} C_VEL
LIN {X 0,Y 602.029,Z 1180.542,A -85,B 0,C 180,E1 26172.106,E2 26172.106} C_VEL
LIN {X 0,Y 603.138,Z 1166.718,A -85,B 0,C 180,E1 26169.931,E2 26169.931} C_VEL
LIN {X 0,Y 604.242,Z 1153.857,A -85,B 0,C 180,E1 26168.177,E2 26168.177} C_VEL
LIN {X 0,Y 605.581,Z 1138.731,A -85,B 0,C 180,E1 26166.402,E2 26166.402} C_VEL
LIN {X 0,Y 607.087,Z 1121.435,A -85,B 0,C 180,E1 26164.646,E2 26164.646} C_VEL
LIN {X 0,Y 608.655,Z 1104.084,A -85,B 0,C 180,E1 26163.091,E2 26163.091} C_VEL
LIN {X 0,Y 610.414,Z 1084.031,A -85,B 0,C 180,E1 26161.533,E2 26161.533} C_VEL
LIN {X 0,Y 611.818,Z 1067.331,A -85,B 0,C 180,E1 26160.395,E2 26160.395} C_VEL
LIN {X 0,Y 613.598,Z 1044.856,A -85,B 0,C 180,E1 26159.062,E2 26159.062} C_VEL
LIN {X 0,Y 615.067,Z 1025.02,A -85,B 0,C 180,E1 26158.06,E2 26158.06} C_VEL
LIN {X 0,Y 616.59,Z 1002.599,A -85,B 0,C 180,E1 26157.082,E2 26157.082} C_VEL
LIN {X 0,Y 617.902,Z 979.483,A -85,B 0,C 180,E1 26156.26,E2 26156.26} C_VEL
LIN {X 0,Y 619.124,Z 955.42,A -85,B 0,C 180,E1 26155.56,E2 26155.56} C_VEL
LIN {X 0,Y 620.117,Z 931.376,A -85,B 0,C 180,E1 26155.041,E2 26155.041} C_VEL
LIN {X 0,Y 620.847,Z 905.57,A -85,B 0,C 180,E1 26154.635,E2 26154.635} C_VEL
LIN {X 0,Y 625.119,Z 668.396,A -85,B 0,C 180,E1 26151.495,E2 26151.495} C_VEL
LIN {X 0,Y 627.125,Z 559.118,A -85,B 0,C 180,E1 26150.022,E2 26150.022} C_VEL
LIN {X 0,Y 625.028,Z 549.453,A -85,B 0,C 180,E1 26149.737,E2 26149.737} C_VEL
LIN {X 0,Y 618.155,Z 537.806,A -85,B 0,C 180,E1 26149.06,E2 26149.06} C_VEL
LIN {X 0,Y 609.497,Z 517.378,A -85,B 0,C 180,E1 26146.752,E2 26146.752} C_VEL
LIN {X 0,Y 602.108,Z 501.279,A -85,B 0,C 180,E1 26144.758,E2 26144.758} C_VEL
LIN {X 0,Y 601.158,Z 498.497,A -85,B 0,C 180,E1 26144.373,E2 26144.373} C_VEL
LIN {X 0,Y 601.085,Z 498.359,A -85,B 0,C 180,E1 26141.331,E2 26141.331} C_VEL
LIN {X 0,Y 601.135,Z 498.307,A -85,B 0,C 180,E1 26138.226,E2 26138.226} C_VEL
LIN {X 0,Y 601.084,Z 498.34,A -85,B 0,C 180,E1 26135.139,E2 26135.139} C_VEL
LIN {X 0,Y 601.134,Z 498.318,A -85,B 0,C 180,E1 26131.934,E2 26131.934} C_VEL
LIN {X 0,Y 601.087,Z 498.345,A -85,B 0,C 180,E1 26128.952,E2 26128.952} C_VEL
LIN {X 0,Y 601.138,Z 498.346,A -85,B 0,C 180,E1 26125.836,E2 26125.836} C_VEL
LIN {X 0,Y 601.09,Z 498.353,A -85,B 0,C 180,E1 26122.701,E2 26122.701} C_VEL
LIN {X 0,Y 601.135,Z 498.348,A -85,B 0,C 180,E1 26119.532,E2 26119.532} C_VEL
LIN {X 0,Y 601.095,Z 498.342,A -85,B 0,C 180,E1 26116.427,E2 26116.427} C_VEL
LIN {X 0,Y 601.123,Z 498.338,A -85,B 0,C 180,E1 26113.172,E2 26113.172} C_VEL
LIN {X 0,Y 601.111,Z 498.349,A -85,B 0,C 180,E1 26110.035,E2 26110.035} C_VEL
LIN {X 0,Y 601.103,Z 498.352,A -85,B 0,C 180,E1 26106.687,E2 26106.687} C_VEL
LIN {X 0,Y 601.132,Z 498.332,A -85,B 0,C 180,E1 26103.528,E2 26103.528} C_VEL
LIN {X 0,Y 601.097,Z 498.347,A -85,B 0,C 180,E1 26100.286,E2 26100.286} C_VEL
LIN {X 0,Y 601.135,Z 498.345,A -85,B 0,C 180,E1 26097.14,E2 26097.14} C_VEL
LIN {X 0,Y 601.097,Z 498.339,A -85,B 0,C 180,E1 26093.984,E2 26093.984} C_VEL
LIN {X 0,Y 601.134,Z 498.349,A -85,B 0,C 180,E1 26090.908,E2 26090.908} C_VEL
LIN {X 0,Y 601.101,Z 498.352,A -85,B 0,C 180,E1 26087.706,E2 26087.706} C_VEL
LIN {X 0,Y 601.133,Z 498.336,A -85,B 0,C 180,E1 26084.566,E2 26084.566} C_VEL
LIN {X 0,Y 601.107,Z 498.338,A -85,B 0,C 180,E1 26081.375,E2 26081.375} C_VEL
LIN {X 0,Y 601.136,Z 498.345,A -85,B 0,C 180,E1 26078.125,E2 26078.125} C_VEL
LIN {X 0,Y 601.126,Z 498.349,A -85,B 0,C 180,E1 26074.902,E2 26074.902} C_VEL
LIN {X 0,Y 601.112,Z 498.355,A -85,B 0,C 180,E1 26071.593,E2 26071.593} C_VEL
LIN {X 0,Y 601.136,Z 498.348,A -85,B 0,C 180,E1 26068.402,E2 26068.402} C_VEL
LIN {X 0,Y 601.108,Z 498.355,A -85,B 0,C 180,E1 26065.211,E2 26065.211} C_VEL
LIN {X 0,Y 601.125,Z 498.302,A -85,B 0,C 180,E1 26062.015,E2 26062.015} C_VEL
LIN {X 0,Y 601.107,Z 498.346,A -85,B 0,C 180,E1 26058.895,E2 26058.895} C_VEL
LIN {X 0,Y 601.129,Z 498.326,A -85,B 0,C 180,E1 26055.661,E2 26055.661} C_VEL
LIN {X 0,Y 601.185,Z 498.794,A -85,B 0,C 180,E1 26055.124,E2 26055.124} C_VEL
LIN {X 0,Y 609.517,Z 517.812,A -85,B 0,C 180,E1 26052.699,E2 26052.699} C_VEL
LIN {X 0,Y 617.811,Z 538.196,A -85,B 0,C 180,E1 26050.334,E2 26050.334} C_VEL
LIN {X 0,Y 621.33,Z 547.643,A -85,B 0,C 180,E1 26049.31,E2 26049.31} C_VEL
LIN {X 0,Y 618.028,Z 593.635,A -85,B 0,C 180,E1 26046.007,E2 26046.007} C_VEL
LIN {X 0,Y 617.533,Z 600.721,A -85,B 0,C 180,E1 26045.507,E2 26045.507} C_VEL
LIN {X 0,Y 616.243,Z 607.105,A -85,B 0,C 180,E1 26045.114,E2 26045.114} C_VEL
LIN {X 0,Y 609.665,Z 624.886,A -85,B 0,C 180,E1 26044.213,E2 26044.213} C_VEL
LIN {X 0,Y 608.667,Z 630.364,A -85,B 0,C 180,E1 26043.868,E2 26043.868} C_VEL
LIN {X 0,Y 608.128,Z 640.918,A -85,B 0,C 180,E1 26043.153,E2 26043.153} C_VEL
LIN {X 0,Y 614.914,Z 679.637,A -85,B 0,C 180,E1 26042.171,E2 26042.171} C_VEL
LIN {X 0,Y 611.719,Z 953.592,A -85,B 0,C 180,E1 26038.905,E2 26038.905} C_VEL
LIN {X 0,Y 610.878,Z 975.869,A -85,B 0,C 180,E1 26038.491,E2 26038.491} C_VEL
LIN {X 0,Y 609.791,Z 996.864,A -85,B 0,C 180,E1 26037.939,E2 26037.939} C_VEL
LIN {X 0,Y 608.341,Z 1017.298,A -85,B 0,C 180,E1 26037.226,E2 26037.226} C_VEL
LIN {X 0,Y 606.665,Z 1038.019,A -85,B 0,C 180,E1 26036.317,E2 26036.317} C_VEL
LIN {X 0,Y 604.959,Z 1056.387,A -85,B 0,C 180,E1 26035.345,E2 26035.345} C_VEL
LIN {X 0,Y 603.061,Z 1074.736,A -85,B 0,C 180,E1 26034.175,E2 26034.175} C_VEL
LIN {X 0,Y 601.087,Z 1092.966,A -85,B 0,C 180,E1 26032.804,E2 26032.804} C_VEL
LIN {X 0,Y 599.233,Z 1109.625,A -85,B 0,C 180,E1 26031.33,E2 26031.33} C_VEL
LIN {X 0,Y 597.509,Z 1124.693,A -85,B 0,C 180,E1 26029.756,E2 26029.756} C_VEL
LIN {X 0,Y 595.894,Z 1139.627,A -85,B 0,C 180,E1 26027.934,E2 26027.934} C_VEL
LIN {X 0,Y 594.635,Z 1152.446,A -85,B 0,C 180,E1 26026.108,E2 26026.108} C_VEL
LIN {X 0,Y 593.599,Z 1164.1,A -85,B 0,C 180,E1 26024.137,E2 26024.137} C_VEL
LIN {X 0,Y 592.861,Z 1174.359,A -85,B 0,C 180,E1 26022.071,E2 26022.071} C_VEL
LIN {X 0,Y 592.4,Z 1182.847,A -85,B 0,C 180,E1 26020.011,E2 26020.011} C_VEL
LIN {X 0,Y 592.118,Z 1189.552,A -85,B 0,C 180,E1 26017.959,E2 26017.959} C_VEL
LIN {X 0,Y 591.974,Z 1194.886,A -85,B 0,C 180,E1 26015.805,E2 26015.805} C_VEL
LIN {X 0,Y 591.931,Z 1198.543,A -85,B 0,C 180,E1 26013.68,E2 26013.68} C_VEL
LIN {X 0,Y 591.915,Z 1200.46,A -85,B 0,C 180,E1 26011.646,E2 26011.646} C_VEL
LIN {X 0,Y 591.908,Z 1200.904,A -85,B 0,C 180,E1 26009.419,E2 26009.419} C_VEL
LIN {X 0,Y 591.923,Z 1199.753,A -85,B 0,C 180,E1 26007.289,E2 26007.289} C_VEL
LIN {X 0,Y 591.943,Z 1197.039,A -85,B 0,C 180,E1 26005.252,E2 26005.252} C_VEL
LIN {X 0,Y 592.024,Z 1192.635,A -85,B 0,C 180,E1 26003.113,E2 26003.113} C_VEL
LIN {X 0,Y 592.235,Z 1186.676,A -85,B 0,C 180,E1 26000.997,E2 26000.997} C_VEL
LIN {X 0,Y 592.596,Z 1178.975,A -85,B 0,C 180,E1 25998.91,E2 25998.91} C_VEL
LIN {X 0,Y 593.179,Z 1169.656,A -85,B 0,C 180,E1 25996.847,E2 25996.847} C_VEL
LIN {X 0,Y 594.033,Z 1159.057,A -85,B 0,C 180,E1 25994.877,E2 25994.877} C_VEL
LIN {X 0,Y 595.195,Z 1146.478,A -85,B 0,C 180,E1 25992.919,E2 25992.919} C_VEL
LIN {X 0,Y 596.594,Z 1132.975,A -85,B 0,C 180,E1 25991.128,E2 25991.128} C_VEL
LIN {X 0,Y 598.235,Z 1118.293,A -85,B 0,C 180,E1 25989.453,E2 25989.453} C_VEL
LIN {X 0,Y 599.957,Z 1103.102,A -85,B 0,C 180,E1 25987.977,E2 25987.977} C_VEL
LIN {X 0,Y 601.846,Z 1085.993,A -85,B 0,C 180,E1 25986.554,E2 25986.554} C_VEL
LIN {X 0,Y 603.794,Z 1068.097,A -85,B 0,C 180,E1 25985.284,E2 25985.284} C_VEL
LIN {X 0,Y 605.559,Z 1050.014,A -85,B 0,C 180,E1 25984.21,E2 25984.21} C_VEL
LIN {X 0,Y 607.398,Z 1029.393,A -85,B 0,C 180,E1 25983.19,E2 25983.19} C_VEL
LIN {X 0,Y 608.914,Z 1010.22,A -85,B 0,C 180,E1 25982.416,E2 25982.416} C_VEL
LIN {X 0,Y 610.194,Z 989.21,A -85,B 0,C 180,E1 25981.752,E2 25981.752} C_VEL
LIN {X 0,Y 611.265,Z 967.152,A -85,B 0,C 180,E1 25981.234,E2 25981.234} C_VEL
LIN {X 0,Y 611.92,Z 945.58,A -85,B 0,C 180,E1 25980.895,E2 25980.895} C_VEL
LIN {X 0,Y 614.904,Z 678.341,A -85,B 0,C 180,E1 25977.717,E2 25977.717} C_VEL
